ABB RAPID module: 05908a28.mod

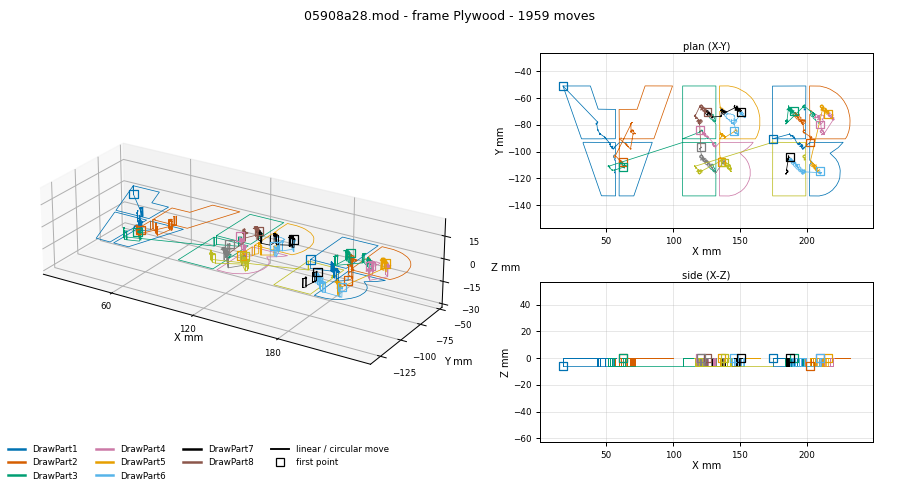
[picture p0: tool path of 05908a28.mod in frame Plywood, 1959 of 1961 moves have a stored position in this frame; points joined in program order, loops and branches not executed]
MODULE ImageDraw
  ! Generated 2026-10-07 09:04 for ABB GoFa CRB 15000-5/0.95: 148 strokes
  ! Page 250 x 180 mm. Work object Plywood: Z points DOWN, so pen-up is -Z and the tool uses orientation [1,0,0,0].
  ! Uses the tool 'tcp' and work object 'Plywood' that already exist on the controller.
  CONST robtarget pOrigin:=[[0,0,0],[1,0,0,0],[0,0,0,0],[9E9,9E9,9E9,9E9,9E9,9E9]];
  CONST jointtarget jHome:=[[0,0,0,0,30,0],[9E9,9E9,9E9,9E9,9E9,9E9]];
  CONST speeddata vTravel:=[250,200,5000,1000];

  PROC DrawImage()
    SingArea\Wrist;
    ConfL\Off;
    ConfJ\Off;
    MoveAbsJ jHome\NoEOffs,vTravel,fine,tcp;
    DrawPart1;
    DrawPart2;
    DrawPart3;
    DrawPart4;
    DrawPart5;
    DrawPart6;
    DrawPart7;
    DrawPart8;
    DrawPart9;
    DrawPart10;
    DrawPart11;
    DrawPart12;
    DrawPart13;
    DrawPart14;
    DrawPart15;
    DrawPart16;
    DrawPart17;
    MoveAbsJ jHome\NoEOffs,vTravel,fine,tcp;
  ENDPROC

  PROC DrawPart1()
    MoveL Offs(pOrigin,17.65,-50.83,-6.00),vTravel,z5,tcp\WObj:=Plywood;
    MoveL Offs(pOrigin,17.65,-50.83,-0.00),v60,z0,tcp\WObj:=Plywood;
    MoveL Offs(pOrigin,38.15,-50.83,-0.00),v40,z0,tcp\WObj:=Plywood;
    MoveL Offs(pOrigin,44.00,-68.18,-0.00),v40,z0,tcp\WObj:=Plywood;
    MoveL Offs(pOrigin,57.00,-68.38,-0.00),v40,z0,tcp\WObj:=Plywood;
    MoveL Offs(pOrigin,56.85,-90.32,-0.00),v40,z0,tcp\WObj:=Plywood;
    MoveL Offs(pOrigin,48.20,-90.38,-0.00),v40,z0,tcp\WObj:=Plywood;
    MoveL Offs(pOrigin,47.75,-90.07,-0.00),v40,z0,tcp\WObj:=Plywood;
    MoveL Offs(pOrigin,47.00,-90.38,-0.00),v40,z0,tcp\WObj:=Plywood;
    MoveL Offs(pOrigin,31.55,-90.38,-0.00),v40,z0,tcp\WObj:=Plywood;
    MoveL Offs(pOrigin,17.65,-50.83,-0.00),v40,fine,tcp\WObj:=Plywood;
    MoveL Offs(pOrigin,17.65,-50.83,-6.00),v60,z5,tcp\WObj:=Plywood;
    MoveL Offs(pOrigin,43.55,-77.82,-6.00),vTravel,z5,tcp\WObj:=Plywood;
    MoveL Offs(pOrigin,43.55,-77.82,-0.00),v60,z0,tcp\WObj:=Plywood;
    MoveL Offs(pOrigin,43.00,-78.68,-0.00),v40,z0,tcp\WObj:=Plywood;
    MoveL Offs(pOrigin,43.85,-77.82,-0.00),v40,z0,tcp\WObj:=Plywood;
    MoveL Offs(pOrigin,43.55,-77.82,-0.00),v40,fine,tcp\WObj:=Plywood;
    MoveL Offs(pOrigin,43.55,-77.82,-6.00),v60,z5,tcp\WObj:=Plywood;
    MoveL Offs(pOrigin,42.95,-78.97,-6.00),vTravel,z5,tcp\WObj:=Plywood;
    MoveL Offs(pOrigin,42.95,-78.97,-0.00),v60,z0,tcp\WObj:=Plywood;
    MoveL Offs(pOrigin,42.65,-78.82,-0.00),v40,z0,tcp\WObj:=Plywood;
    MoveL Offs(pOrigin,42.35,-79.12,-0.00),v40,z0,tcp\WObj:=Plywood;
    MoveL Offs(pOrigin,42.50,-79.43,-0.00),v40,z0,tcp\WObj:=Plywood;
    MoveL Offs(pOrigin,42.95,-78.97,-0.00),v40,z0,tcp\WObj:=Plywood;
    MoveL Offs(pOrigin,42.65,-78.82,-0.00),v40,z0,tcp\WObj:=Plywood;
    MoveL Offs(pOrigin,42.35,-79.28,-0.00),v40,z0,tcp\WObj:=Plywood;
    MoveL Offs(pOrigin,42.95,-78.97,-0.00),v40,fine,tcp\WObj:=Plywood;
    MoveL Offs(pOrigin,42.95,-78.97,-6.00),v60,z5,tcp\WObj:=Plywood;
    MoveL Offs(pOrigin,43.55,-83.78,-6.00),vTravel,z5,tcp\WObj:=Plywood;
    MoveL Offs(pOrigin,43.55,-83.78,-0.00),v60,z0,tcp\WObj:=Plywood;
    MoveL Offs(pOrigin,44.15,-83.78,-0.00),v40,z0,tcp\WObj:=Plywood;
    MoveL Offs(pOrigin,43.55,-83.78,-0.00),v40,fine,tcp\WObj:=Plywood;
    MoveL Offs(pOrigin,43.55,-83.78,-6.00),v60,z5,tcp\WObj:=Plywood;
    MoveL Offs(pOrigin,45.35,-86.62,-6.00),vTravel,z5,tcp\WObj:=Plywood;
    MoveL Offs(pOrigin,45.35,-86.62,-0.00),v60,z0,tcp\WObj:=Plywood;
    MoveL Offs(pOrigin,45.20,-87.07,-0.00),v40,z0,tcp\WObj:=Plywood;
    MoveL Offs(pOrigin,45.65,-86.78,-0.00),v40,z0,tcp\WObj:=Plywood;
    MoveL Offs(pOrigin,45.35,-86.62,-0.00),v40,z0,tcp\WObj:=Plywood;
    MoveL Offs(pOrigin,45.05,-86.93,-0.00),v40,z0,tcp\WObj:=Plywood;
    MoveL Offs(pOrigin,45.35,-87.07,-0.00),v40,z0,tcp\WObj:=Plywood;
    MoveL Offs(pOrigin,45.65,-86.78,-0.00),v40,z0,tcp\WObj:=Plywood;
    MoveL Offs(pOrigin,45.35,-86.62,-0.00),v40,fine,tcp\WObj:=Plywood;
    MoveL Offs(pOrigin,45.35,-86.62,-6.00),v60,z5,tcp\WObj:=Plywood;
    MoveL Offs(pOrigin,48.80,-89.03,-6.00),vTravel,z5,tcp\WObj:=Plywood;
    MoveL Offs(pOrigin,48.80,-89.03,-0.00),v60,z0,tcp\WObj:=Plywood;
    MoveL Offs(pOrigin,48.80,-89.47,-0.00),v40,z0,tcp\WObj:=Plywood;
    MoveL Offs(pOrigin,49.10,-89.32,-0.00),v40,z0,tcp\WObj:=Plywood;
    MoveL Offs(pOrigin,48.95,-89.03,-0.00),v40,z0,tcp\WObj:=Plywood;
    MoveL Offs(pOrigin,48.65,-89.32,-0.00),v40,z0,tcp\WObj:=Plywood;
    MoveL Offs(pOrigin,48.95,-89.47,-0.00),v40,z0,tcp\WObj:=Plywood;
    MoveL Offs(pOrigin,49.10,-89.18,-0.00),v40,z0,tcp\WObj:=Plywood;
    MoveL Offs(pOrigin,48.80,-89.03,-0.00),v40,fine,tcp\WObj:=Plywood;
    MoveL Offs(pOrigin,48.80,-89.03,-6.00),v60,z5,tcp\WObj:=Plywood;
    MoveL Offs(pOrigin,53.00,-94.12,-6.00),vTravel,z5,tcp\WObj:=Plywood;
    MoveL Offs(pOrigin,53.00,-94.12,-0.00),v60,z0,tcp\WObj:=Plywood;
    MoveL Offs(pOrigin,52.55,-94.57,-0.00),v40,z0,tcp\WObj:=Plywood;
    MoveL Offs(pOrigin,52.85,-94.72,-0.00),v40,z0,tcp\WObj:=Plywood;
    MoveL Offs(pOrigin,53.15,-94.28,-0.00),v40,z0,tcp\WObj:=Plywood;
    MoveL Offs(pOrigin,52.55,-94.57,-0.00),v40,z0,tcp\WObj:=Plywood;
    MoveL Offs(pOrigin,52.85,-94.72,-0.00),v40,z0,tcp\WObj:=Plywood;
    MoveL Offs(pOrigin,53.15,-94.43,-0.00),v40,z0,tcp\WObj:=Plywood;
    MoveL Offs(pOrigin,53.00,-94.12,-0.00),v40,fine,tcp\WObj:=Plywood;
    MoveL Offs(pOrigin,53.00,-94.12,-6.00),v60,z5,tcp\WObj:=Plywood;
    MoveL Offs(pOrigin,53.00,-95.93,-6.00),vTravel,z5,tcp\WObj:=Plywood;
    MoveL Offs(pOrigin,53.00,-95.93,-0.00),v60,z0,tcp\WObj:=Plywood;
    MoveL Offs(pOrigin,53.60,-95.93,-0.00),v40,z0,tcp\WObj:=Plywood;
    MoveL Offs(pOrigin,53.00,-95.93,-0.00),v40,fine,tcp\WObj:=Plywood;
    MoveL Offs(pOrigin,53.00,-95.93,-6.00),v60,z5,tcp\WObj:=Plywood;
    MoveL Offs(pOrigin,54.40,-96.53,-6.00),vTravel,z5,tcp\WObj:=Plywood;
    MoveL Offs(pOrigin,54.40,-96.53,-0.00),v60,z0,tcp\WObj:=Plywood;
    MoveL Offs(pOrigin,55.10,-95.82,-0.00),v40,z0,tcp\WObj:=Plywood;
    MoveL Offs(pOrigin,54.65,-95.93,-0.00),v40,z0,tcp\WObj:=Plywood;
    MoveL Offs(pOrigin,54.40,-96.53,-0.00),v40,z0,tcp\WObj:=Plywood;
    MoveL Offs(pOrigin,54.35,-97.43,-0.00),v40,z0,tcp\WObj:=Plywood;
    MoveL Offs(pOrigin,54.35,-96.97,-0.00),v40,z0,tcp\WObj:=Plywood;
    MoveL Offs(pOrigin,54.35,-97.43,-0.00),v40,z0,tcp\WObj:=Plywood;
    MoveL Offs(pOrigin,54.90,-97.72,-0.00),v40,z0,tcp\WObj:=Plywood;
    MoveL Offs(pOrigin,55.25,-98.12,-0.00),v40,z0,tcp\WObj:=Plywood;
    MoveL Offs(pOrigin,55.65,-97.88,-0.00),v40,z0,tcp\WObj:=Plywood;
    MoveL Offs(pOrigin,55.40,-97.57,-0.00),v40,z0,tcp\WObj:=Plywood;
    MoveL Offs(pOrigin,54.90,-97.72,-0.00),v40,fine,tcp\WObj:=Plywood;
    MoveL Offs(pOrigin,54.90,-97.72,-6.00),v60,z5,tcp\WObj:=Plywood;
    MoveL Offs(pOrigin,56.00,-97.12,-6.00),vTravel,z5,tcp\WObj:=Plywood;
    MoveL Offs(pOrigin,56.00,-97.12,-0.00),v60,z0,tcp\WObj:=Plywood;
    MoveL Offs(pOrigin,56.30,-97.38,-0.00),v40,z0,tcp\WObj:=Plywood;
    MoveL Offs(pOrigin,56.90,-96.97,-0.00),v40,z0,tcp\WObj:=Plywood;
    MoveL Offs(pOrigin,56.90,-102.07,-0.00),v40,z0,tcp\WObj:=Plywood;
    MoveL Offs(pOrigin,55.75,-102.68,-0.00),v40,z0,tcp\WObj:=Plywood;
    MoveL Offs(pOrigin,55.40,-103.88,-0.00),v40,z0,tcp\WObj:=Plywood;
    MoveL Offs(pOrigin,55.85,-104.62,-0.00),v40,z0,tcp\WObj:=Plywood;
    MoveL Offs(pOrigin,56.90,-105.07,-0.00),v40,z0,tcp\WObj:=Plywood;
    MoveL Offs(pOrigin,56.15,-106.12,-0.00),v40,z0,tcp\WObj:=Plywood;
    MoveL Offs(pOrigin,56.30,-106.38,-0.00),v40,z0,tcp\WObj:=Plywood;
    MoveL Offs(pOrigin,56.90,-106.28,-0.00),v40,z0,tcp\WObj:=Plywood;
    MoveL Offs(pOrigin,56.90,-113.78,-0.00),v40,z0,tcp\WObj:=Plywood;
    MoveL Offs(pOrigin,56.40,-113.93,-0.00),v40,z0,tcp\WObj:=Plywood;
    MoveL Offs(pOrigin,56.90,-114.68,-0.00),v40,z0,tcp\WObj:=Plywood;
    MoveL Offs(pOrigin,56.70,-115.22,-0.00),v40,z0,tcp\WObj:=Plywood;
    MoveL Offs(pOrigin,56.20,-114.97,-0.00),v40,z0,tcp\WObj:=Plywood;
    MoveL Offs(pOrigin,56.10,-115.88,-0.00),v40,z0,tcp\WObj:=Plywood;
    MoveL Offs(pOrigin,56.85,-115.62,-0.00),v40,z0,tcp\WObj:=Plywood;
    MoveL Offs(pOrigin,57.05,-116.03,-0.00),v40,z0,tcp\WObj:=Plywood;
    MoveL Offs(pOrigin,57.00,-133.07,-0.00),v40,z0,tcp\WObj:=Plywood;
    MoveL Offs(pOrigin,46.45,-132.98,-0.00),v40,z0,tcp\WObj:=Plywood;
    MoveL Offs(pOrigin,32.70,-93.53,-0.00),v40,z0,tcp\WObj:=Plywood;
    MoveL Offs(pOrigin,32.75,-92.97,-0.00),v40,z0,tcp\WObj:=Plywood;
    MoveL Offs(pOrigin,56.90,-93.12,-0.00),v40,z0,tcp\WObj:=Plywood;
    MoveL Offs(pOrigin,56.90,-95.93,-0.00),v40,z0,tcp\WObj:=Plywood;
    MoveL Offs(pOrigin,56.70,-96.32,-0.00),v40,z0,tcp\WObj:=Plywood;
    MoveL Offs(pOrigin,56.20,-96.38,-0.00),v40,z0,tcp\WObj:=Plywood;
    MoveL Offs(pOrigin,56.00,-97.12,-0.00),v40,fine,tcp\WObj:=Plywood;
    MoveL Offs(pOrigin,56.00,-97.12,-6.00),v60,z5,tcp\WObj:=Plywood;
    MoveL Offs(pOrigin,59.80,-93.12,-6.00),vTravel,z5,tcp\WObj:=Plywood;
    MoveL Offs(pOrigin,59.80,-93.12,-0.00),v60,z0,tcp\WObj:=Plywood;
    MoveL Offs(pOrigin,84.45,-92.97,-0.00),v40,z0,tcp\WObj:=Plywood;
    MoveL Offs(pOrigin,70.65,-133.07,-0.00),v40,z0,tcp\WObj:=Plywood;
    MoveL Offs(pOrigin,59.65,-133.07,-0.00),v40,z0,tcp\WObj:=Plywood;
    MoveL Offs(pOrigin,59.75,-108.97,-0.00),v40,z0,tcp\WObj:=Plywood;
    MoveL Offs(pOrigin,60.20,-109.28,-0.00),v40,z0,tcp\WObj:=Plywood;
    MoveL Offs(pOrigin,60.95,-109.18,-0.00),v40,z0,tcp\WObj:=Plywood;
  ENDPROC

  PROC DrawPart2()
    MoveL Offs(pOrigin,62.25,-107.93,-0.00),v40,z0,tcp\WObj:=Plywood;
    MoveL Offs(pOrigin,61.25,-106.72,-0.00),v40,z0,tcp\WObj:=Plywood;
    MoveL Offs(pOrigin,60.65,-106.57,-0.00),v40,z0,tcp\WObj:=Plywood;
    MoveL Offs(pOrigin,60.25,-106.88,-0.00),v40,z0,tcp\WObj:=Plywood;
    MoveL Offs(pOrigin,60.20,-107.62,-0.00),v40,z0,tcp\WObj:=Plywood;
    MoveL Offs(pOrigin,60.75,-108.68,-0.00),v40,z0,tcp\WObj:=Plywood;
    MoveL Offs(pOrigin,59.75,-108.22,-0.00),v40,z0,tcp\WObj:=Plywood;
    MoveL Offs(pOrigin,59.75,-105.93,-0.00),v40,z0,tcp\WObj:=Plywood;
    MoveL Offs(pOrigin,59.90,-106.28,-0.00),v40,z0,tcp\WObj:=Plywood;
    MoveL Offs(pOrigin,60.25,-106.12,-0.00),v40,z0,tcp\WObj:=Plywood;
    MoveL Offs(pOrigin,59.75,-105.22,-0.00),v40,z0,tcp\WObj:=Plywood;
    MoveL Offs(pOrigin,59.80,-93.12,-0.00),v40,fine,tcp\WObj:=Plywood;
    MoveL Offs(pOrigin,59.80,-93.12,-6.00),v60,z5,tcp\WObj:=Plywood;
    MoveL Offs(pOrigin,59.80,-90.32,-6.00),vTravel,z5,tcp\WObj:=Plywood;
    MoveL Offs(pOrigin,59.80,-90.32,-0.00),v60,z0,tcp\WObj:=Plywood;
    MoveL Offs(pOrigin,59.65,-68.38,-0.00),v40,z0,tcp\WObj:=Plywood;
    MoveL Offs(pOrigin,73.10,-68.28,-0.00),v40,z0,tcp\WObj:=Plywood;
    MoveL Offs(pOrigin,79.10,-50.78,-0.00),v40,z0,tcp\WObj:=Plywood;
    MoveL Offs(pOrigin,99.60,-50.83,-0.00),v40,z0,tcp\WObj:=Plywood;
    MoveL Offs(pOrigin,85.65,-90.32,-0.00),v40,z0,tcp\WObj:=Plywood;
    MoveL Offs(pOrigin,61.25,-90.38,-0.00),v40,z0,tcp\WObj:=Plywood;
    MoveL Offs(pOrigin,61.25,-89.68,-0.00),v40,z0,tcp\WObj:=Plywood;
    MoveL Offs(pOrigin,59.80,-90.32,-0.00),v40,fine,tcp\WObj:=Plywood;
    MoveL Offs(pOrigin,59.80,-90.32,-6.00),v60,z5,tcp\WObj:=Plywood;
    MoveL Offs(pOrigin,64.40,-94.12,-6.00),vTravel,z5,tcp\WObj:=Plywood;
    MoveL Offs(pOrigin,64.40,-94.12,-0.00),v60,z0,tcp\WObj:=Plywood;
    MoveL Offs(pOrigin,65.00,-94.12,-0.00),v40,z0,tcp\WObj:=Plywood;
    MoveL Offs(pOrigin,64.40,-94.12,-0.00),v40,z0,tcp\WObj:=Plywood;
    MoveL Offs(pOrigin,65.00,-95.03,-0.00),v40,z0,tcp\WObj:=Plywood;
    MoveL Offs(pOrigin,65.30,-95.32,-0.00),v40,z0,tcp\WObj:=Plywood;
    MoveL Offs(pOrigin,65.60,-95.18,-0.00),v40,z0,tcp\WObj:=Plywood;
    MoveL Offs(pOrigin,65.45,-94.57,-0.00),v40,z0,tcp\WObj:=Plywood;
    MoveL Offs(pOrigin,65.00,-95.03,-0.00),v40,z0,tcp\WObj:=Plywood;
    MoveL Offs(pOrigin,65.30,-95.32,-0.00),v40,z0,tcp\WObj:=Plywood;
    MoveL Offs(pOrigin,65.60,-95.18,-0.00),v40,z0,tcp\WObj:=Plywood;
    MoveL Offs(pOrigin,65.45,-94.57,-0.00),v40,z0,tcp\WObj:=Plywood;
    MoveL Offs(pOrigin,65.00,-95.03,-0.00),v40,fine,tcp\WObj:=Plywood;
    MoveL Offs(pOrigin,65.00,-95.03,-6.00),v60,z5,tcp\WObj:=Plywood;
    MoveL Offs(pOrigin,65.90,-95.93,-6.00),vTravel,z5,tcp\WObj:=Plywood;
    MoveL Offs(pOrigin,65.90,-95.93,-0.00),v60,z0,tcp\WObj:=Plywood;
    MoveL Offs(pOrigin,66.50,-95.93,-0.00),v40,z0,tcp\WObj:=Plywood;
    MoveL Offs(pOrigin,65.90,-95.93,-0.00),v40,fine,tcp\WObj:=Plywood;
    MoveL Offs(pOrigin,65.90,-95.93,-6.00),v60,z5,tcp\WObj:=Plywood;
    MoveL Offs(pOrigin,68.15,-97.88,-6.00),vTravel,z5,tcp\WObj:=Plywood;
    MoveL Offs(pOrigin,68.15,-97.88,-0.00),v60,z0,tcp\WObj:=Plywood;
    MoveL Offs(pOrigin,68.45,-98.03,-0.00),v40,z0,tcp\WObj:=Plywood;
    MoveL Offs(pOrigin,68.60,-97.72,-0.00),v40,z0,tcp\WObj:=Plywood;
    MoveL Offs(pOrigin,68.15,-97.88,-0.00),v40,z0,tcp\WObj:=Plywood;
    MoveL Offs(pOrigin,68.45,-98.03,-0.00),v40,z0,tcp\WObj:=Plywood;
    MoveL Offs(pOrigin,68.45,-97.57,-0.00),v40,z0,tcp\WObj:=Plywood;
    MoveL Offs(pOrigin,68.15,-97.88,-0.00),v40,fine,tcp\WObj:=Plywood;
    MoveL Offs(pOrigin,68.15,-97.88,-6.00),v60,z5,tcp\WObj:=Plywood;
    MoveL Offs(pOrigin,70.10,-86.78,-6.00),vTravel,z5,tcp\WObj:=Plywood;
    MoveL Offs(pOrigin,70.10,-86.78,-0.00),v60,z0,tcp\WObj:=Plywood;
    MoveL Offs(pOrigin,70.55,-86.32,-0.00),v40,z0,tcp\WObj:=Plywood;
    MoveL Offs(pOrigin,70.25,-86.18,-0.00),v40,z0,tcp\WObj:=Plywood;
    MoveL Offs(pOrigin,69.95,-86.62,-0.00),v40,z0,tcp\WObj:=Plywood;
    MoveL Offs(pOrigin,70.55,-86.32,-0.00),v40,z0,tcp\WObj:=Plywood;
    MoveL Offs(pOrigin,70.25,-86.18,-0.00),v40,z0,tcp\WObj:=Plywood;
    MoveL Offs(pOrigin,69.95,-86.47,-0.00),v40,z0,tcp\WObj:=Plywood;
    MoveL Offs(pOrigin,70.10,-86.78,-0.00),v40,fine,tcp\WObj:=Plywood;
    MoveL Offs(pOrigin,70.10,-86.78,-6.00),v60,z5,tcp\WObj:=Plywood;
    MoveL Offs(pOrigin,71.45,-86.47,-6.00),vTravel,z5,tcp\WObj:=Plywood;
    MoveL Offs(pOrigin,71.45,-86.47,-0.00),v60,z0,tcp\WObj:=Plywood;
    MoveL Offs(pOrigin,71.75,-86.62,-0.00),v40,z0,tcp\WObj:=Plywood;
    MoveL Offs(pOrigin,71.90,-86.32,-0.00),v40,z0,tcp\WObj:=Plywood;
    MoveL Offs(pOrigin,71.45,-86.47,-0.00),v40,z0,tcp\WObj:=Plywood;
    MoveL Offs(pOrigin,71.75,-86.62,-0.00),v40,z0,tcp\WObj:=Plywood;
    MoveL Offs(pOrigin,71.75,-86.18,-0.00),v40,z0,tcp\WObj:=Plywood;
    MoveL Offs(pOrigin,71.45,-86.47,-0.00),v40,fine,tcp\WObj:=Plywood;
    MoveL Offs(pOrigin,71.45,-86.47,-6.00),v60,z5,tcp\WObj:=Plywood;
    MoveL Offs(pOrigin,70.50,-84.97,-6.00),vTravel,z5,tcp\WObj:=Plywood;
    MoveL Offs(pOrigin,70.50,-84.97,-0.00),v60,z0,tcp\WObj:=Plywood;
    MoveL Offs(pOrigin,70.50,-84.22,-0.00),v40,z0,tcp\WObj:=Plywood;
    MoveL Offs(pOrigin,69.95,-83.68,-0.00),v40,z0,tcp\WObj:=Plywood;
    MoveL Offs(pOrigin,69.35,-83.62,-0.00),v40,z0,tcp\WObj:=Plywood;
    MoveL Offs(pOrigin,68.75,-84.07,-0.00),v40,z0,tcp\WObj:=Plywood;
    MoveL Offs(pOrigin,68.90,-84.32,-0.00),v40,z0,tcp\WObj:=Plywood;
    MoveL Offs(pOrigin,69.80,-84.03,-0.00),v40,z0,tcp\WObj:=Plywood;
    MoveL Offs(pOrigin,70.50,-84.97,-0.00),v40,fine,tcp\WObj:=Plywood;
    MoveL Offs(pOrigin,70.50,-84.97,-6.00),v60,z5,tcp\WObj:=Plywood;
    MoveL Offs(pOrigin,68.60,-85.47,-6.00),vTravel,z5,tcp\WObj:=Plywood;
    MoveL Offs(pOrigin,68.60,-85.47,-0.00),v60,z0,tcp\WObj:=Plywood;
    MoveL Offs(pOrigin,68.45,-84.47,-0.00),v40,z0,tcp\WObj:=Plywood;
    MoveL Offs(pOrigin,68.15,-84.97,-0.00),v40,z0,tcp\WObj:=Plywood;
    MoveL Offs(pOrigin,68.60,-85.47,-0.00),v40,fine,tcp\WObj:=Plywood;
    MoveL Offs(pOrigin,68.60,-85.47,-6.00),v60,z5,tcp\WObj:=Plywood;
    MoveL Offs(pOrigin,68.45,-79.28,-6.00),vTravel,z5,tcp\WObj:=Plywood;
    MoveL Offs(pOrigin,68.45,-79.28,-0.00),v60,z0,tcp\WObj:=Plywood;
    MoveL Offs(pOrigin,68.75,-78.97,-0.00),v40,z0,tcp\WObj:=Plywood;
    MoveL Offs(pOrigin,68.45,-78.82,-0.00),v40,z0,tcp\WObj:=Plywood;
    MoveL Offs(pOrigin,68.30,-79.28,-0.00),v40,z0,tcp\WObj:=Plywood;
    MoveL Offs(pOrigin,68.75,-78.97,-0.00),v40,z0,tcp\WObj:=Plywood;
    MoveL Offs(pOrigin,68.45,-78.82,-0.00),v40,z0,tcp\WObj:=Plywood;
    MoveL Offs(pOrigin,68.15,-79.12,-0.00),v40,z0,tcp\WObj:=Plywood;
    MoveL Offs(pOrigin,68.45,-79.28,-0.00),v40,fine,tcp\WObj:=Plywood;
    MoveL Offs(pOrigin,68.45,-79.28,-6.00),v60,z5,tcp\WObj:=Plywood;
    MoveL Offs(pOrigin,69.20,-78.07,-6.00),vTravel,z5,tcp\WObj:=Plywood;
    MoveL Offs(pOrigin,69.20,-78.07,-0.00),v60,z0,tcp\WObj:=Plywood;
    MoveL Offs(pOrigin,69.65,-78.07,-0.00),v40,z0,tcp\WObj:=Plywood;
    MoveL Offs(pOrigin,69.20,-78.07,-0.00),v40,fine,tcp\WObj:=Plywood;
    MoveL Offs(pOrigin,69.20,-78.07,-6.00),v60,z5,tcp\WObj:=Plywood;
    MoveL Offs(pOrigin,56.90,-102.97,-6.00),vTravel,z5,tcp\WObj:=Plywood;
    MoveL Offs(pOrigin,56.90,-102.97,-0.00),v60,z0,tcp\WObj:=Plywood;
    MoveL Offs(pOrigin,56.85,-104.43,-0.00),v40,z0,tcp\WObj:=Plywood;
    MoveL Offs(pOrigin,55.85,-103.88,-0.00),v40,z0,tcp\WObj:=Plywood;
    MoveL Offs(pOrigin,55.90,-103.18,-0.00),v40,z0,tcp\WObj:=Plywood;
    MoveL Offs(pOrigin,56.60,-102.82,-0.00),v40,z0,tcp\WObj:=Plywood;
    MoveL Offs(pOrigin,56.90,-102.97,-0.00),v40,fine,tcp\WObj:=Plywood;
    MoveL Offs(pOrigin,56.90,-102.97,-6.00),v60,z5,tcp\WObj:=Plywood;
    MoveL Offs(pOrigin,60.80,-107.22,-6.00),vTravel,z5,tcp\WObj:=Plywood;
    MoveL Offs(pOrigin,60.80,-107.22,-0.00),v60,z0,tcp\WObj:=Plywood;
    MoveL Offs(pOrigin,61.35,-107.47,-0.00),v40,z0,tcp\WObj:=Plywood;
    MoveL Offs(pOrigin,61.25,-108.12,-0.00),v40,z0,tcp\WObj:=Plywood;
    MoveL Offs(pOrigin,60.70,-107.78,-0.00),v40,z0,tcp\WObj:=Plywood;
    MoveL Offs(pOrigin,60.80,-107.22,-0.00),v40,fine,tcp\WObj:=Plywood;
    MoveL Offs(pOrigin,60.80,-107.22,-6.00),v60,z5,tcp\WObj:=Plywood;
    MoveL Offs(pOrigin,62.75,-108.57,-6.00),vTravel,z5,tcp\WObj:=Plywood;
    MoveL Offs(pOrigin,62.75,-108.57,-0.00),v60,z0,tcp\WObj:=Plywood;
    MoveL Offs(pOrigin,61.20,-110.03,-0.00),v40,z0,tcp\WObj:=Plywood;
  ENDPROC

  PROC DrawPart3()
    MoveL Offs(pOrigin,62.45,-111.22,-0.00),v40,z0,tcp\WObj:=Plywood;
    MoveL Offs(pOrigin,63.60,-110.32,-0.00),v40,z0,tcp\WObj:=Plywood;
    MoveL Offs(pOrigin,63.35,-110.12,-0.00),v40,z0,tcp\WObj:=Plywood;
    MoveL Offs(pOrigin,62.45,-110.78,-0.00),v40,z0,tcp\WObj:=Plywood;
    MoveL Offs(pOrigin,62.05,-110.47,-0.00),v40,z0,tcp\WObj:=Plywood;
    MoveL Offs(pOrigin,62.05,-109.72,-0.00),v40,z0,tcp\WObj:=Plywood;
    MoveL Offs(pOrigin,62.85,-108.82,-0.00),v40,z0,tcp\WObj:=Plywood;
    MoveL Offs(pOrigin,62.75,-108.57,-0.00),v40,fine,tcp\WObj:=Plywood;
    MoveL Offs(pOrigin,62.75,-108.57,-6.00),v60,z5,tcp\WObj:=Plywood;
    MoveL Offs(pOrigin,63.80,-109.72,-6.00),vTravel,z5,tcp\WObj:=Plywood;
    MoveL Offs(pOrigin,63.80,-109.72,-0.00),v60,z0,tcp\WObj:=Plywood;
    MoveL Offs(pOrigin,63.50,-110.03,-0.00),v40,z0,tcp\WObj:=Plywood;
    MoveL Offs(pOrigin,63.80,-110.18,-0.00),v40,z0,tcp\WObj:=Plywood;
    MoveL Offs(pOrigin,63.95,-109.88,-0.00),v40,z0,tcp\WObj:=Plywood;
    MoveL Offs(pOrigin,63.50,-110.03,-0.00),v40,z0,tcp\WObj:=Plywood;
    MoveL Offs(pOrigin,63.80,-110.18,-0.00),v40,z0,tcp\WObj:=Plywood;
    MoveL Offs(pOrigin,63.80,-109.72,-0.00),v40,z0,tcp\WObj:=Plywood;
    MoveL Offs(pOrigin,64.40,-110.47,-0.00),v40,z0,tcp\WObj:=Plywood;
    MoveL Offs(pOrigin,63.85,-111.22,-0.00),v40,z0,tcp\WObj:=Plywood;
    MoveL Offs(pOrigin,64.85,-110.88,-0.00),v40,z0,tcp\WObj:=Plywood;
    MoveL Offs(pOrigin,65.10,-110.18,-0.00),v40,z0,tcp\WObj:=Plywood;
    MoveL Offs(pOrigin,64.40,-110.47,-0.00),v40,z0,tcp\WObj:=Plywood;
    MoveL Offs(pOrigin,63.80,-111.32,-0.00),v40,z0,tcp\WObj:=Plywood;
    MoveL Offs(pOrigin,63.15,-111.97,-0.00),v40,z0,tcp\WObj:=Plywood;
    MoveL Offs(pOrigin,63.65,-112.32,-0.00),v40,z0,tcp\WObj:=Plywood;
    MoveL Offs(pOrigin,63.80,-111.32,-0.00),v40,fine,tcp\WObj:=Plywood;
    MoveL Offs(pOrigin,63.80,-111.32,-6.00),v60,z5,tcp\WObj:=Plywood;
    MoveL Offs(pOrigin,56.00,-113.78,-6.00),vTravel,z5,tcp\WObj:=Plywood;
    MoveL Offs(pOrigin,56.00,-113.78,-0.00),v60,z0,tcp\WObj:=Plywood;
    MoveL Offs(pOrigin,56.45,-113.78,-0.00),v40,z0,tcp\WObj:=Plywood;
    MoveL Offs(pOrigin,56.00,-113.78,-0.00),v40,fine,tcp\WObj:=Plywood;
    MoveL Offs(pOrigin,56.00,-113.78,-6.00),v60,z5,tcp\WObj:=Plywood;
    MoveL Offs(pOrigin,54.35,-113.78,-6.00),vTravel,z5,tcp\WObj:=Plywood;
    MoveL Offs(pOrigin,54.35,-113.78,-0.00),v60,z0,tcp\WObj:=Plywood;
    MoveL Offs(pOrigin,54.80,-113.78,-0.00),v40,z0,tcp\WObj:=Plywood;
    MoveL Offs(pOrigin,54.35,-113.78,-0.00),v40,fine,tcp\WObj:=Plywood;
    MoveL Offs(pOrigin,54.35,-113.78,-6.00),v60,z5,tcp\WObj:=Plywood;
    MoveL Offs(pOrigin,52.70,-112.18,-6.00),vTravel,z5,tcp\WObj:=Plywood;
    MoveL Offs(pOrigin,52.70,-112.18,-0.00),v60,z0,tcp\WObj:=Plywood;
    MoveL Offs(pOrigin,52.70,-111.32,-0.00),v40,z0,tcp\WObj:=Plywood;
    MoveL Offs(pOrigin,52.70,-112.18,-0.00),v40,fine,tcp\WObj:=Plywood;
    MoveL Offs(pOrigin,52.70,-112.18,-6.00),v60,z5,tcp\WObj:=Plywood;
    MoveL Offs(pOrigin,51.65,-110.93,-6.00),vTravel,z5,tcp\WObj:=Plywood;
    MoveL Offs(pOrigin,51.65,-110.93,-0.00),v60,z0,tcp\WObj:=Plywood;
    MoveL Offs(pOrigin,51.95,-110.47,-0.00),v40,z0,tcp\WObj:=Plywood;
    MoveL Offs(pOrigin,51.35,-110.78,-0.00),v40,z0,tcp\WObj:=Plywood;
    MoveL Offs(pOrigin,51.65,-110.93,-0.00),v40,z0,tcp\WObj:=Plywood;
    MoveL Offs(pOrigin,51.95,-110.62,-0.00),v40,z0,tcp\WObj:=Plywood;
    MoveL Offs(pOrigin,51.80,-110.32,-0.00),v40,z0,tcp\WObj:=Plywood;
    MoveL Offs(pOrigin,51.35,-110.78,-0.00),v40,z0,tcp\WObj:=Plywood;
    MoveL Offs(pOrigin,51.65,-110.93,-0.00),v40,fine,tcp\WObj:=Plywood;
    MoveL Offs(pOrigin,51.65,-110.93,-6.00),v60,z5,tcp\WObj:=Plywood;
    MoveL Offs(pOrigin,107.20,-93.07,-6.00),vTravel,z5,tcp\WObj:=Plywood;
    MoveL Offs(pOrigin,107.20,-93.07,-0.00),v60,z0,tcp\WObj:=Plywood;
    MoveL Offs(pOrigin,132.00,-93.12,-0.00),v40,z0,tcp\WObj:=Plywood;
    MoveL Offs(pOrigin,132.05,-113.32,-0.00),v40,z0,tcp\WObj:=Plywood;
    MoveL Offs(pOrigin,130.70,-114.32,-0.00),v40,z0,tcp\WObj:=Plywood;
    MoveL Offs(pOrigin,130.30,-114.22,-0.00),v40,z0,tcp\WObj:=Plywood;
    MoveL Offs(pOrigin,130.30,-113.62,-0.00),v40,z0,tcp\WObj:=Plywood;
    MoveL Offs(pOrigin,131.30,-112.43,-0.00),v40,z0,tcp\WObj:=Plywood;
    MoveL Offs(pOrigin,130.60,-112.07,-0.00),v40,z0,tcp\WObj:=Plywood;
    MoveL Offs(pOrigin,130.00,-110.62,-0.00),v40,z0,tcp\WObj:=Plywood;
    MoveL Offs(pOrigin,130.20,-109.72,-0.00),v40,z0,tcp\WObj:=Plywood;
    MoveL Offs(pOrigin,129.65,-109.28,-0.00),v40,z0,tcp\WObj:=Plywood;
    MoveL Offs(pOrigin,127.30,-111.97,-0.00),v40,z0,tcp\WObj:=Plywood;
    MoveL Offs(pOrigin,128.45,-113.22,-0.00),v40,z0,tcp\WObj:=Plywood;
    MoveL Offs(pOrigin,129.45,-113.28,-0.00),v40,z0,tcp\WObj:=Plywood;
    MoveL Offs(pOrigin,129.40,-113.93,-0.00),v40,z0,tcp\WObj:=Plywood;
    MoveL Offs(pOrigin,130.40,-115.03,-0.00),v40,z0,tcp\WObj:=Plywood;
    MoveL Offs(pOrigin,130.85,-115.07,-0.00),v40,z0,tcp\WObj:=Plywood;
    MoveL Offs(pOrigin,131.90,-114.18,-0.00),v40,z0,tcp\WObj:=Plywood;
    MoveL Offs(pOrigin,132.05,-114.38,-0.00),v40,z0,tcp\WObj:=Plywood;
    MoveL Offs(pOrigin,131.45,-114.97,-0.00),v40,z0,tcp\WObj:=Plywood;
    MoveL Offs(pOrigin,131.45,-116.03,-0.00),v40,z0,tcp\WObj:=Plywood;
    MoveL Offs(pOrigin,132.05,-116.78,-0.00),v40,z0,tcp\WObj:=Plywood;
    MoveL Offs(pOrigin,132.00,-133.07,-0.00),v40,z0,tcp\WObj:=Plywood;
    MoveL Offs(pOrigin,107.15,-133.07,-0.00),v40,z0,tcp\WObj:=Plywood;
    MoveL Offs(pOrigin,107.20,-93.07,-0.00),v40,fine,tcp\WObj:=Plywood;
    MoveL Offs(pOrigin,107.20,-93.07,-6.00),v60,z5,tcp\WObj:=Plywood;
    MoveL Offs(pOrigin,107.20,-90.32,-6.00),vTravel,z5,tcp\WObj:=Plywood;
    MoveL Offs(pOrigin,107.20,-90.32,-0.00),v60,z0,tcp\WObj:=Plywood;
    MoveL Offs(pOrigin,107.20,-50.83,-0.00),v40,z0,tcp\WObj:=Plywood;
    MoveL Offs(pOrigin,132.05,-50.83,-0.00),v40,z0,tcp\WObj:=Plywood;
    MoveL Offs(pOrigin,132.05,-75.82,-0.00),v40,z0,tcp\WObj:=Plywood;
    MoveL Offs(pOrigin,130.70,-76.82,-0.00),v40,z0,tcp\WObj:=Plywood;
    MoveL Offs(pOrigin,130.35,-76.72,-0.00),v40,z0,tcp\WObj:=Plywood;
    MoveL Offs(pOrigin,130.30,-76.12,-0.00),v40,z0,tcp\WObj:=Plywood;
    MoveL Offs(pOrigin,131.30,-74.93,-0.00),v40,z0,tcp\WObj:=Plywood;
    MoveL Offs(pOrigin,130.55,-74.47,-0.00),v40,z0,tcp\WObj:=Plywood;
    MoveL Offs(pOrigin,129.90,-72.97,-0.00),v40,z0,tcp\WObj:=Plywood;
    MoveL Offs(pOrigin,130.35,-72.68,-0.00),v40,z0,tcp\WObj:=Plywood;
    MoveL Offs(pOrigin,129.80,-71.93,-0.00),v40,z0,tcp\WObj:=Plywood;
    MoveL Offs(pOrigin,128.45,-72.97,-0.00),v40,z0,tcp\WObj:=Plywood;
    MoveL Offs(pOrigin,127.25,-74.47,-0.00),v40,z0,tcp\WObj:=Plywood;
    MoveL Offs(pOrigin,128.45,-75.72,-0.00),v40,z0,tcp\WObj:=Plywood;
    MoveL Offs(pOrigin,129.45,-75.78,-0.00),v40,z0,tcp\WObj:=Plywood;
    MoveL Offs(pOrigin,129.40,-76.43,-0.00),v40,z0,tcp\WObj:=Plywood;
    MoveL Offs(pOrigin,130.40,-77.57,-0.00),v40,z0,tcp\WObj:=Plywood;
    MoveL Offs(pOrigin,131.00,-77.57,-0.00),v40,z0,tcp\WObj:=Plywood;
    MoveL Offs(pOrigin,132.05,-76.72,-0.00),v40,z0,tcp\WObj:=Plywood;
    MoveL Offs(pOrigin,131.30,-78.07,-0.00),v40,z0,tcp\WObj:=Plywood;
    MoveL Offs(pOrigin,132.05,-79.43,-0.00),v40,z0,tcp\WObj:=Plywood;
    MoveL Offs(pOrigin,132.00,-90.32,-0.00),v40,z0,tcp\WObj:=Plywood;
    MoveL Offs(pOrigin,125.60,-90.28,-0.00),v40,z0,tcp\WObj:=Plywood;
    MoveL Offs(pOrigin,125.80,-89.78,-0.00),v40,z0,tcp\WObj:=Plywood;
    MoveL Offs(pOrigin,125.45,-89.47,-0.00),v40,z0,tcp\WObj:=Plywood;
    MoveL Offs(pOrigin,124.25,-90.38,-0.00),v40,z0,tcp\WObj:=Plywood;
    MoveL Offs(pOrigin,107.20,-90.32,-0.00),v40,fine,tcp\WObj:=Plywood;
    MoveL Offs(pOrigin,107.20,-90.32,-6.00),v60,z5,tcp\WObj:=Plywood;
    MoveL Offs(pOrigin,120.05,-85.32,-6.00),vTravel,z5,tcp\WObj:=Plywood;
    MoveL Offs(pOrigin,120.05,-85.32,-0.00),v60,z0,tcp\WObj:=Plywood;
    MoveL Offs(pOrigin,120.05,-84.62,-0.00),v40,z0,tcp\WObj:=Plywood;
    MoveL Offs(pOrigin,120.05,-85.32,-0.00),v40,fine,tcp\WObj:=Plywood;
    MoveL Offs(pOrigin,120.05,-85.32,-6.00),v60,z5,tcp\WObj:=Plywood;
    MoveL Offs(pOrigin,120.50,-84.18,-6.00),vTravel,z5,tcp\WObj:=Plywood;
    MoveL Offs(pOrigin,120.50,-84.18,-0.00),v60,z0,tcp\WObj:=Plywood;
    MoveL Offs(pOrigin,121.55,-84.12,-0.00),v40,z0,tcp\WObj:=Plywood;
    MoveL Offs(pOrigin,121.85,-84.97,-0.00),v40,z0,tcp\WObj:=Plywood;
    MoveL Offs(pOrigin,122.25,-84.82,-0.00),v40,z0,tcp\WObj:=Plywood;
    MoveL Offs(pOrigin,121.55,-83.68,-0.00),v40,z0,tcp\WObj:=Plywood;
  ENDPROC

  PROC DrawPart4()
    MoveL Offs(pOrigin,120.40,-83.93,-0.00),v40,z0,tcp\WObj:=Plywood;
    MoveL Offs(pOrigin,120.50,-84.18,-0.00),v40,fine,tcp\WObj:=Plywood;
    MoveL Offs(pOrigin,120.50,-84.18,-6.00),v60,z5,tcp\WObj:=Plywood;
    MoveL Offs(pOrigin,122.30,-85.57,-6.00),vTravel,z5,tcp\WObj:=Plywood;
    MoveL Offs(pOrigin,122.30,-85.57,-0.00),v60,z0,tcp\WObj:=Plywood;
    MoveL Offs(pOrigin,121.85,-86.43,-0.00),v40,z0,tcp\WObj:=Plywood;
    MoveL Offs(pOrigin,122.40,-86.18,-0.00),v40,z0,tcp\WObj:=Plywood;
    MoveL Offs(pOrigin,122.90,-85.32,-0.00),v40,z0,tcp\WObj:=Plywood;
    MoveL Offs(pOrigin,122.30,-85.57,-0.00),v40,z0,tcp\WObj:=Plywood;
    MoveL Offs(pOrigin,122.75,-86.47,-0.00),v40,z0,tcp\WObj:=Plywood;
    MoveL Offs(pOrigin,122.20,-87.38,-0.00),v40,z0,tcp\WObj:=Plywood;
    MoveL Offs(pOrigin,123.00,-87.07,-0.00),v40,z0,tcp\WObj:=Plywood;
    MoveL Offs(pOrigin,123.20,-86.38,-0.00),v40,z0,tcp\WObj:=Plywood;
    MoveL Offs(pOrigin,122.75,-86.47,-0.00),v40,z0,tcp\WObj:=Plywood;
    MoveL Offs(pOrigin,123.20,-87.07,-0.00),v40,z0,tcp\WObj:=Plywood;
    MoveL Offs(pOrigin,123.05,-87.38,-0.00),v40,z0,tcp\WObj:=Plywood;
    MoveL Offs(pOrigin,123.50,-87.82,-0.00),v40,z0,tcp\WObj:=Plywood;
    MoveL Offs(pOrigin,123.65,-87.53,-0.00),v40,z0,tcp\WObj:=Plywood;
    MoveL Offs(pOrigin,123.05,-87.22,-0.00),v40,z0,tcp\WObj:=Plywood;
    MoveL Offs(pOrigin,123.50,-87.82,-0.00),v40,z0,tcp\WObj:=Plywood;
    MoveL Offs(pOrigin,123.65,-87.53,-0.00),v40,z0,tcp\WObj:=Plywood;
    MoveL Offs(pOrigin,123.20,-87.07,-0.00),v40,z0,tcp\WObj:=Plywood;
    MoveL Offs(pOrigin,123.80,-86.68,-0.00),v40,z0,tcp\WObj:=Plywood;
    MoveL Offs(pOrigin,124.20,-86.62,-0.00),v40,z0,tcp\WObj:=Plywood;
    MoveL Offs(pOrigin,123.95,-86.28,-0.00),v40,z0,tcp\WObj:=Plywood;
    MoveL Offs(pOrigin,123.55,-86.32,-0.00),v40,z0,tcp\WObj:=Plywood;
    MoveL Offs(pOrigin,123.80,-86.68,-0.00),v40,z0,tcp\WObj:=Plywood;
    MoveL Offs(pOrigin,124.10,-86.78,-0.00),v40,z0,tcp\WObj:=Plywood;
    MoveL Offs(pOrigin,124.40,-87.38,-0.00),v40,z0,tcp\WObj:=Plywood;
    MoveL Offs(pOrigin,124.55,-86.93,-0.00),v40,z0,tcp\WObj:=Plywood;
    MoveL Offs(pOrigin,124.25,-86.62,-0.00),v40,z0,tcp\WObj:=Plywood;
    MoveL Offs(pOrigin,124.40,-87.38,-0.00),v40,z0,tcp\WObj:=Plywood;
    MoveL Offs(pOrigin,124.55,-86.93,-0.00),v40,z0,tcp\WObj:=Plywood;
    MoveL Offs(pOrigin,124.10,-86.78,-0.00),v40,z0,tcp\WObj:=Plywood;
    MoveL Offs(pOrigin,123.80,-87.82,-0.00),v40,z0,tcp\WObj:=Plywood;
    MoveL Offs(pOrigin,123.55,-87.82,-0.00),v40,z0,tcp\WObj:=Plywood;
    MoveL Offs(pOrigin,123.50,-88.38,-0.00),v40,z0,tcp\WObj:=Plywood;
    MoveL Offs(pOrigin,123.95,-88.28,-0.00),v40,z0,tcp\WObj:=Plywood;
    MoveL Offs(pOrigin,123.80,-87.82,-0.00),v40,fine,tcp\WObj:=Plywood;
    MoveL Offs(pOrigin,123.80,-87.82,-6.00),v60,z5,tcp\WObj:=Plywood;
    MoveL Offs(pOrigin,124.70,-88.72,-6.00),vTravel,z5,tcp\WObj:=Plywood;
    MoveL Offs(pOrigin,124.70,-88.72,-0.00),v60,z0,tcp\WObj:=Plywood;
    MoveL Offs(pOrigin,125.75,-88.38,-0.00),v40,z0,tcp\WObj:=Plywood;
    MoveL Offs(pOrigin,125.75,-88.12,-0.00),v40,z0,tcp\WObj:=Plywood;
    MoveL Offs(pOrigin,125.15,-87.93,-0.00),v40,z0,tcp\WObj:=Plywood;
    MoveL Offs(pOrigin,124.70,-88.72,-0.00),v40,fine,tcp\WObj:=Plywood;
    MoveL Offs(pOrigin,124.70,-88.72,-6.00),v60,z5,tcp\WObj:=Plywood;
    MoveL Offs(pOrigin,126.10,-88.88,-6.00),vTravel,z5,tcp\WObj:=Plywood;
    MoveL Offs(pOrigin,126.10,-88.88,-0.00),v60,z0,tcp\WObj:=Plywood;
    MoveL Offs(pOrigin,125.95,-89.47,-0.00),v40,z0,tcp\WObj:=Plywood;
    MoveL Offs(pOrigin,126.60,-89.03,-0.00),v40,z0,tcp\WObj:=Plywood;
    MoveL Offs(pOrigin,126.10,-88.88,-0.00),v40,fine,tcp\WObj:=Plywood;
    MoveL Offs(pOrigin,126.10,-88.88,-6.00),v60,z5,tcp\WObj:=Plywood;
    MoveL Offs(pOrigin,129.95,-93.28,-6.00),vTravel,z5,tcp\WObj:=Plywood;
    MoveL Offs(pOrigin,129.95,-93.28,-0.00),v60,z0,tcp\WObj:=Plywood;
    MoveL Offs(pOrigin,129.20,-94.22,-0.00),v40,z0,tcp\WObj:=Plywood;
    MoveL Offs(pOrigin,129.65,-94.12,-0.00),v40,z0,tcp\WObj:=Plywood;
    MoveL Offs(pOrigin,130.20,-93.38,-0.00),v40,z0,tcp\WObj:=Plywood;
    MoveL Offs(pOrigin,129.95,-93.28,-0.00),v40,z0,tcp\WObj:=Plywood;
    MoveL Offs(pOrigin,130.55,-93.82,-0.00),v40,z0,tcp\WObj:=Plywood;
    MoveL Offs(pOrigin,130.70,-94.12,-0.00),v40,z0,tcp\WObj:=Plywood;
    MoveL Offs(pOrigin,131.00,-93.68,-0.00),v40,z0,tcp\WObj:=Plywood;
    MoveL Offs(pOrigin,130.55,-93.82,-0.00),v40,z0,tcp\WObj:=Plywood;
    MoveL Offs(pOrigin,130.70,-94.12,-0.00),v40,z0,tcp\WObj:=Plywood;
    MoveL Offs(pOrigin,131.00,-93.82,-0.00),v40,z0,tcp\WObj:=Plywood;
    MoveL Offs(pOrigin,130.85,-93.53,-0.00),v40,z0,tcp\WObj:=Plywood;
    MoveL Offs(pOrigin,130.55,-93.82,-0.00),v40,z0,tcp\WObj:=Plywood;
    MoveL Offs(pOrigin,130.40,-93.97,-0.00),v40,z0,tcp\WObj:=Plywood;
    MoveL Offs(pOrigin,130.40,-94.43,-0.00),v40,z0,tcp\WObj:=Plywood;
    MoveL Offs(pOrigin,130.70,-94.12,-0.00),v40,z0,tcp\WObj:=Plywood;
    MoveL Offs(pOrigin,130.40,-93.97,-0.00),v40,z0,tcp\WObj:=Plywood;
    MoveL Offs(pOrigin,130.25,-94.28,-0.00),v40,z0,tcp\WObj:=Plywood;
    MoveL Offs(pOrigin,130.70,-94.12,-0.00),v40,z0,tcp\WObj:=Plywood;
    MoveL Offs(pOrigin,130.40,-93.97,-0.00),v40,z0,tcp\WObj:=Plywood;
    MoveL Offs(pOrigin,130.10,-94.72,-0.00),v40,z0,tcp\WObj:=Plywood;
    MoveL Offs(pOrigin,129.80,-94.57,-0.00),v40,z0,tcp\WObj:=Plywood;
    MoveL Offs(pOrigin,129.80,-95.18,-0.00),v40,z0,tcp\WObj:=Plywood;
    MoveL Offs(pOrigin,130.10,-94.72,-0.00),v40,z0,tcp\WObj:=Plywood;
    MoveL Offs(pOrigin,129.80,-94.57,-0.00),v40,z0,tcp\WObj:=Plywood;
    MoveL Offs(pOrigin,129.65,-95.03,-0.00),v40,z0,tcp\WObj:=Plywood;
    MoveL Offs(pOrigin,130.10,-94.72,-0.00),v40,fine,tcp\WObj:=Plywood;
    MoveL Offs(pOrigin,130.10,-94.72,-6.00),v60,z5,tcp\WObj:=Plywood;
    MoveL Offs(pOrigin,130.40,-95.93,-6.00),vTravel,z5,tcp\WObj:=Plywood;
    MoveL Offs(pOrigin,130.40,-95.93,-0.00),v60,z0,tcp\WObj:=Plywood;
    MoveL Offs(pOrigin,131.00,-95.93,-0.00),v40,z0,tcp\WObj:=Plywood;
    MoveL Offs(pOrigin,130.40,-95.93,-0.00),v40,fine,tcp\WObj:=Plywood;
    MoveL Offs(pOrigin,130.40,-95.93,-6.00),v60,z5,tcp\WObj:=Plywood;
    MoveL Offs(pOrigin,131.45,-95.32,-6.00),vTravel,z5,tcp\WObj:=Plywood;
    MoveL Offs(pOrigin,131.45,-95.32,-0.00),v60,z0,tcp\WObj:=Plywood;
    MoveL Offs(pOrigin,131.75,-95.47,-0.00),v40,z0,tcp\WObj:=Plywood;
    MoveL Offs(pOrigin,131.90,-95.18,-0.00),v40,z0,tcp\WObj:=Plywood;
    MoveL Offs(pOrigin,131.45,-95.18,-0.00),v40,z0,tcp\WObj:=Plywood;
    MoveL Offs(pOrigin,131.75,-95.47,-0.00),v40,z0,tcp\WObj:=Plywood;
    MoveL Offs(pOrigin,131.75,-95.03,-0.00),v40,z0,tcp\WObj:=Plywood;
    MoveL Offs(pOrigin,131.45,-95.32,-0.00),v40,z0,tcp\WObj:=Plywood;
    MoveL Offs(pOrigin,131.75,-96.47,-0.00),v40,z0,tcp\WObj:=Plywood;
    MoveL Offs(pOrigin,131.45,-96.82,-0.00),v40,z0,tcp\WObj:=Plywood;
    MoveL Offs(pOrigin,131.75,-97.47,-0.00),v40,z0,tcp\WObj:=Plywood;
    MoveL Offs(pOrigin,131.75,-96.47,-0.00),v40,fine,tcp\WObj:=Plywood;
    MoveL Offs(pOrigin,131.75,-96.47,-6.00),v60,z5,tcp\WObj:=Plywood;
    MoveL Offs(pOrigin,134.90,-93.12,-6.00),vTravel,z5,tcp\WObj:=Plywood;
    MoveL Offs(pOrigin,134.90,-93.12,-0.00),v60,z0,tcp\WObj:=Plywood;
    MoveL Offs(pOrigin,159.95,-92.97,-0.00),v40,z0,tcp\WObj:=Plywood;
    MoveL Offs(pOrigin,158.45,-94.88,-0.00),v40,z0,tcp\WObj:=Plywood;
    MoveL Offs(pOrigin,155.30,-97.72,-0.00),v40,z0,tcp\WObj:=Plywood;
    MoveL Offs(pOrigin,150.15,-101.18,-0.00),v40,z0,tcp\WObj:=Plywood;
    MoveL Offs(pOrigin,153.95,-104.78,-0.00),v40,z0,tcp\WObj:=Plywood;
    MoveL Offs(pOrigin,155.15,-106.43,-0.00),v40,z0,tcp\WObj:=Plywood;
    MoveL Offs(pOrigin,156.55,-109.12,-0.00),v40,z0,tcp\WObj:=Plywood;
    MoveL Offs(pOrigin,157.70,-113.32,-0.00),v40,z0,tcp\WObj:=Plywood;
    MoveL Offs(pOrigin,157.70,-117.97,-0.00),v40,z0,tcp\WObj:=Plywood;
    MoveL Offs(pOrigin,156.85,-121.28,-0.00),v40,z0,tcp\WObj:=Plywood;
    MoveL Offs(pOrigin,155.20,-124.72,-0.00),v40,z0,tcp\WObj:=Plywood;
    MoveL Offs(pOrigin,153.35,-127.28,-0.00),v40,z0,tcp\WObj:=Plywood;
    MoveL Offs(pOrigin,150.95,-129.52,-0.00),v40,z0,tcp\WObj:=Plywood;
    MoveL Offs(pOrigin,146.30,-132.12,-0.00),v40,z0,tcp\WObj:=Plywood;
    MoveL Offs(pOrigin,141.95,-133.12,-0.00),v40,z0,tcp\WObj:=Plywood;
    MoveL Offs(pOrigin,134.75,-133.07,-0.00),v40,z0,tcp\WObj:=Plywood;
    MoveL Offs(pOrigin,134.90,-106.53,-0.00),v40,z0,tcp\WObj:=Plywood;
    MoveL Offs(pOrigin,135.20,-107.18,-0.00),v40,z0,tcp\WObj:=Plywood;
  ENDPROC

  PROC DrawPart5()
    MoveL Offs(pOrigin,136.25,-107.47,-0.00),v40,z0,tcp\WObj:=Plywood;
    MoveL Offs(pOrigin,137.10,-106.72,-0.00),v40,z0,tcp\WObj:=Plywood;
    MoveL Offs(pOrigin,136.15,-105.53,-0.00),v40,z0,tcp\WObj:=Plywood;
    MoveL Offs(pOrigin,136.85,-105.62,-0.00),v40,z0,tcp\WObj:=Plywood;
    MoveL Offs(pOrigin,137.15,-106.53,-0.00),v40,z0,tcp\WObj:=Plywood;
    MoveL Offs(pOrigin,137.60,-106.12,-0.00),v40,z0,tcp\WObj:=Plywood;
    MoveL Offs(pOrigin,137.00,-105.07,-0.00),v40,z0,tcp\WObj:=Plywood;
    MoveL Offs(pOrigin,136.25,-104.78,-0.00),v40,z0,tcp\WObj:=Plywood;
    MoveL Offs(pOrigin,135.00,-105.72,-0.00),v40,z0,tcp\WObj:=Plywood;
    MoveL Offs(pOrigin,135.85,-104.32,-0.00),v40,z0,tcp\WObj:=Plywood;
    MoveL Offs(pOrigin,135.50,-104.12,-0.00),v40,z0,tcp\WObj:=Plywood;
    MoveL Offs(pOrigin,134.95,-104.43,-0.00),v40,z0,tcp\WObj:=Plywood;
    MoveL Offs(pOrigin,135.20,-103.12,-0.00),v40,z0,tcp\WObj:=Plywood;
    MoveL Offs(pOrigin,134.90,-102.53,-0.00),v40,z0,tcp\WObj:=Plywood;
    MoveL Offs(pOrigin,134.90,-93.12,-0.00),v40,fine,tcp\WObj:=Plywood;
    MoveL Offs(pOrigin,134.90,-93.12,-6.00),v60,z5,tcp\WObj:=Plywood;
    MoveL Offs(pOrigin,134.95,-90.32,-6.00),vTravel,z5,tcp\WObj:=Plywood;
    MoveL Offs(pOrigin,134.95,-90.32,-0.00),v60,z0,tcp\WObj:=Plywood;
    MoveL Offs(pOrigin,134.90,-86.78,-0.00),v40,z0,tcp\WObj:=Plywood;
    MoveL Offs(pOrigin,135.60,-85.57,-0.00),v40,z0,tcp\WObj:=Plywood;
    MoveL Offs(pOrigin,134.90,-85.72,-0.00),v40,z0,tcp\WObj:=Plywood;
    MoveL Offs(pOrigin,135.20,-84.82,-0.00),v40,z0,tcp\WObj:=Plywood;
    MoveL Offs(pOrigin,134.90,-83.47,-0.00),v40,z0,tcp\WObj:=Plywood;
    MoveL Offs(pOrigin,134.95,-74.78,-0.00),v40,z0,tcp\WObj:=Plywood;
    MoveL Offs(pOrigin,135.30,-74.62,-0.00),v40,z0,tcp\WObj:=Plywood;
    MoveL Offs(pOrigin,134.90,-74.03,-0.00),v40,z0,tcp\WObj:=Plywood;
    MoveL Offs(pOrigin,134.90,-69.82,-0.00),v40,z0,tcp\WObj:=Plywood;
    MoveL Offs(pOrigin,136.70,-69.88,-0.00),v40,z0,tcp\WObj:=Plywood;
    MoveL Offs(pOrigin,137.75,-68.47,-0.00),v40,z0,tcp\WObj:=Plywood;
    MoveL Offs(pOrigin,137.15,-67.57,-0.00),v40,z0,tcp\WObj:=Plywood;
    MoveL Offs(pOrigin,136.40,-67.28,-0.00),v40,z0,tcp\WObj:=Plywood;
    MoveL Offs(pOrigin,135.25,-67.68,-0.00),v40,z0,tcp\WObj:=Plywood;
    MoveL Offs(pOrigin,135.80,-66.97,-0.00),v40,z0,tcp\WObj:=Plywood;
    MoveL Offs(pOrigin,135.65,-66.57,-0.00),v40,z0,tcp\WObj:=Plywood;
    MoveL Offs(pOrigin,134.95,-66.93,-0.00),v40,z0,tcp\WObj:=Plywood;
    MoveL Offs(pOrigin,135.20,-66.22,-0.00),v40,z0,tcp\WObj:=Plywood;
    MoveL Offs(pOrigin,134.75,-61.58,-0.00),v40,z0,tcp\WObj:=Plywood;
    MoveL Offs(pOrigin,134.75,-50.83,-0.00),v40,z0,tcp\WObj:=Plywood;
    MoveL Offs(pOrigin,141.35,-50.78,-0.00),v40,z0,tcp\WObj:=Plywood;
    MoveL Offs(pOrigin,146.00,-51.67,-0.00),v40,z0,tcp\WObj:=Plywood;
    MoveL Offs(pOrigin,148.85,-52.67,-0.00),v40,z0,tcp\WObj:=Plywood;
    MoveL Offs(pOrigin,154.55,-55.88,-0.00),v40,z0,tcp\WObj:=Plywood;
    MoveL Offs(pOrigin,158.45,-59.47,-0.00),v40,z0,tcp\WObj:=Plywood;
    MoveL Offs(pOrigin,160.10,-61.58,-0.00),v40,z0,tcp\WObj:=Plywood;
    MoveL Offs(pOrigin,163.00,-66.82,-0.00),v40,z0,tcp\WObj:=Plywood;
    MoveL Offs(pOrigin,164.00,-69.82,-0.00),v40,z0,tcp\WObj:=Plywood;
    MoveL Offs(pOrigin,164.90,-74.32,-0.00),v40,z0,tcp\WObj:=Plywood;
    MoveL Offs(pOrigin,164.90,-80.62,-0.00),v40,z0,tcp\WObj:=Plywood;
    MoveL Offs(pOrigin,164.45,-83.47,-0.00),v40,z0,tcp\WObj:=Plywood;
    MoveL Offs(pOrigin,163.00,-87.97,-0.00),v40,z0,tcp\WObj:=Plywood;
    MoveL Offs(pOrigin,161.60,-90.38,-0.00),v40,z0,tcp\WObj:=Plywood;
    MoveL Offs(pOrigin,138.65,-90.38,-0.00),v40,z0,tcp\WObj:=Plywood;
    MoveL Offs(pOrigin,138.05,-90.07,-0.00),v40,z0,tcp\WObj:=Plywood;
    MoveL Offs(pOrigin,137.30,-90.38,-0.00),v40,z0,tcp\WObj:=Plywood;
    MoveL Offs(pOrigin,134.95,-90.32,-0.00),v40,fine,tcp\WObj:=Plywood;
    MoveL Offs(pOrigin,134.95,-90.32,-6.00),v60,z5,tcp\WObj:=Plywood;
    MoveL Offs(pOrigin,136.55,-88.43,-6.00),vTravel,z5,tcp\WObj:=Plywood;
    MoveL Offs(pOrigin,136.55,-88.43,-0.00),v60,z0,tcp\WObj:=Plywood;
    MoveL Offs(pOrigin,136.85,-88.12,-0.00),v40,z0,tcp\WObj:=Plywood;
    MoveL Offs(pOrigin,136.70,-87.68,-0.00),v40,z0,tcp\WObj:=Plywood;
    MoveL Offs(pOrigin,136.40,-87.82,-0.00),v40,z0,tcp\WObj:=Plywood;
    MoveL Offs(pOrigin,136.55,-88.43,-0.00),v40,z0,tcp\WObj:=Plywood;
    MoveL Offs(pOrigin,136.85,-87.82,-0.00),v40,z0,tcp\WObj:=Plywood;
    MoveL Offs(pOrigin,136.40,-87.82,-0.00),v40,z0,tcp\WObj:=Plywood;
    MoveL Offs(pOrigin,136.55,-88.43,-0.00),v40,z0,tcp\WObj:=Plywood;
    MoveL Offs(pOrigin,136.40,-87.82,-0.00),v40,z0,tcp\WObj:=Plywood;
    MoveL Offs(pOrigin,136.55,-87.53,-0.00),v40,z0,tcp\WObj:=Plywood;
    MoveL Offs(pOrigin,136.10,-87.22,-0.00),v40,z0,tcp\WObj:=Plywood;
    MoveL Offs(pOrigin,136.40,-87.82,-0.00),v40,z0,tcp\WObj:=Plywood;
    MoveL Offs(pOrigin,136.55,-87.53,-0.00),v40,z0,tcp\WObj:=Plywood;
    MoveL Offs(pOrigin,136.25,-87.22,-0.00),v40,z0,tcp\WObj:=Plywood;
    MoveL Offs(pOrigin,135.95,-87.38,-0.00),v40,z0,tcp\WObj:=Plywood;
    MoveL Offs(pOrigin,136.40,-87.82,-0.00),v40,z0,tcp\WObj:=Plywood;
    MoveL Offs(pOrigin,135.80,-87.18,-0.00),v40,z0,tcp\WObj:=Plywood;
    MoveL Offs(pOrigin,136.35,-86.32,-0.00),v40,z0,tcp\WObj:=Plywood;
    MoveL Offs(pOrigin,135.50,-86.47,-0.00),v40,z0,tcp\WObj:=Plywood;
    MoveL Offs(pOrigin,135.40,-87.07,-0.00),v40,z0,tcp\WObj:=Plywood;
    MoveL Offs(pOrigin,135.80,-87.18,-0.00),v40,z0,tcp\WObj:=Plywood;
    MoveL Offs(pOrigin,136.55,-86.38,-0.00),v40,z0,tcp\WObj:=Plywood;
    MoveL Offs(pOrigin,137.40,-87.53,-0.00),v40,z0,tcp\WObj:=Plywood;
    MoveL Offs(pOrigin,137.10,-86.47,-0.00),v40,z0,tcp\WObj:=Plywood;
    MoveL Offs(pOrigin,136.55,-86.38,-0.00),v40,fine,tcp\WObj:=Plywood;
    MoveL Offs(pOrigin,136.55,-86.38,-6.00),v60,z5,tcp\WObj:=Plywood;
    MoveL Offs(pOrigin,137.90,-87.97,-6.00),vTravel,z5,tcp\WObj:=Plywood;
    MoveL Offs(pOrigin,137.90,-87.97,-0.00),v60,z0,tcp\WObj:=Plywood;
    MoveL Offs(pOrigin,137.90,-88.43,-0.00),v40,z0,tcp\WObj:=Plywood;
    MoveL Offs(pOrigin,138.35,-88.12,-0.00),v40,z0,tcp\WObj:=Plywood;
    MoveL Offs(pOrigin,137.90,-87.97,-0.00),v40,z0,tcp\WObj:=Plywood;
    MoveL Offs(pOrigin,137.75,-88.28,-0.00),v40,z0,tcp\WObj:=Plywood;
    MoveL Offs(pOrigin,138.05,-88.43,-0.00),v40,z0,tcp\WObj:=Plywood;
    MoveL Offs(pOrigin,138.35,-88.12,-0.00),v40,z0,tcp\WObj:=Plywood;
    MoveL Offs(pOrigin,137.90,-87.97,-0.00),v40,fine,tcp\WObj:=Plywood;
    MoveL Offs(pOrigin,137.90,-87.97,-6.00),v60,z5,tcp\WObj:=Plywood;
    MoveL Offs(pOrigin,139.10,-88.88,-6.00),vTravel,z5,tcp\WObj:=Plywood;
    MoveL Offs(pOrigin,139.10,-88.88,-0.00),v60,z0,tcp\WObj:=Plywood;
    MoveL Offs(pOrigin,138.80,-89.32,-0.00),v40,z0,tcp\WObj:=Plywood;
    MoveL Offs(pOrigin,139.10,-89.47,-0.00),v40,z0,tcp\WObj:=Plywood;
    MoveL Offs(pOrigin,139.40,-89.18,-0.00),v40,z0,tcp\WObj:=Plywood;
    MoveL Offs(pOrigin,139.10,-88.88,-0.00),v40,z0,tcp\WObj:=Plywood;
    MoveL Offs(pOrigin,138.80,-89.32,-0.00),v40,z0,tcp\WObj:=Plywood;
    MoveL Offs(pOrigin,139.10,-89.47,-0.00),v40,z0,tcp\WObj:=Plywood;
    MoveL Offs(pOrigin,139.40,-89.18,-0.00),v40,z0,tcp\WObj:=Plywood;
    MoveL Offs(pOrigin,139.10,-88.88,-0.00),v40,z0,tcp\WObj:=Plywood;
    MoveL Offs(pOrigin,138.50,-89.47,-0.00),v40,z0,tcp\WObj:=Plywood;
    MoveL Offs(pOrigin,138.20,-89.78,-0.00),v40,z0,tcp\WObj:=Plywood;
    MoveL Offs(pOrigin,138.35,-90.18,-0.00),v40,z0,tcp\WObj:=Plywood;
    MoveL Offs(pOrigin,138.80,-89.78,-0.00),v40,z0,tcp\WObj:=Plywood;
    MoveL Offs(pOrigin,138.50,-89.47,-0.00),v40,fine,tcp\WObj:=Plywood;
    MoveL Offs(pOrigin,138.50,-89.47,-6.00),v60,z5,tcp\WObj:=Plywood;
    MoveL Offs(pOrigin,145.55,-85.12,-6.00),vTravel,z5,tcp\WObj:=Plywood;
    MoveL Offs(pOrigin,145.55,-85.12,-0.00),v60,z0,tcp\WObj:=Plywood;
    MoveL Offs(pOrigin,146.00,-85.72,-0.00),v40,z0,tcp\WObj:=Plywood;
    MoveL Offs(pOrigin,146.25,-85.72,-0.00),v40,z0,tcp\WObj:=Plywood;
    MoveL Offs(pOrigin,146.10,-84.68,-0.00),v40,z0,tcp\WObj:=Plywood;
    MoveL Offs(pOrigin,146.60,-84.12,-0.00),v40,z0,tcp\WObj:=Plywood;
    MoveL Offs(pOrigin,147.35,-84.12,-0.00),v40,z0,tcp\WObj:=Plywood;
    MoveL Offs(pOrigin,147.90,-84.97,-0.00),v40,z0,tcp\WObj:=Plywood;
    MoveL Offs(pOrigin,147.90,-84.22,-0.00),v40,z0,tcp\WObj:=Plywood;
    MoveL Offs(pOrigin,147.20,-83.53,-0.00),v40,z0,tcp\WObj:=Plywood;
    MoveL Offs(pOrigin,146.30,-83.72,-0.00),v40,z0,tcp\WObj:=Plywood;
  ENDPROC

  PROC DrawPart6()
    MoveL Offs(pOrigin,145.60,-84.53,-0.00),v40,z0,tcp\WObj:=Plywood;
    MoveL Offs(pOrigin,145.55,-85.12,-0.00),v40,z0,tcp\WObj:=Plywood;
    MoveL Offs(pOrigin,146.30,-85.88,-0.00),v40,z0,tcp\WObj:=Plywood;
    MoveL Offs(pOrigin,147.05,-85.88,-0.00),v40,z0,tcp\WObj:=Plywood;
    MoveL Offs(pOrigin,146.30,-85.88,-0.00),v40,fine,tcp\WObj:=Plywood;
    MoveL Offs(pOrigin,146.30,-85.88,-6.00),v60,z5,tcp\WObj:=Plywood;
    MoveL Offs(pOrigin,147.35,-86.47,-6.00),vTravel,z5,tcp\WObj:=Plywood;
    MoveL Offs(pOrigin,147.35,-86.47,-0.00),v60,z0,tcp\WObj:=Plywood;
    MoveL Offs(pOrigin,147.80,-86.32,-0.00),v40,z0,tcp\WObj:=Plywood;
    MoveL Offs(pOrigin,147.50,-86.18,-0.00),v40,z0,tcp\WObj:=Plywood;
    MoveL Offs(pOrigin,147.50,-86.62,-0.00),v40,z0,tcp\WObj:=Plywood;
    MoveL Offs(pOrigin,147.80,-86.32,-0.00),v40,z0,tcp\WObj:=Plywood;
    MoveL Offs(pOrigin,147.50,-86.18,-0.00),v40,z0,tcp\WObj:=Plywood;
    MoveL Offs(pOrigin,147.35,-86.47,-0.00),v40,z0,tcp\WObj:=Plywood;
    MoveL Offs(pOrigin,148.25,-86.78,-0.00),v40,z0,tcp\WObj:=Plywood;
    MoveL Offs(pOrigin,148.40,-87.07,-0.00),v40,z0,tcp\WObj:=Plywood;
    MoveL Offs(pOrigin,148.70,-86.93,-0.00),v40,z0,tcp\WObj:=Plywood;
    MoveL Offs(pOrigin,148.55,-86.47,-0.00),v40,z0,tcp\WObj:=Plywood;
    MoveL Offs(pOrigin,148.25,-86.93,-0.00),v40,z0,tcp\WObj:=Plywood;
    MoveL Offs(pOrigin,148.70,-86.93,-0.00),v40,z0,tcp\WObj:=Plywood;
    MoveL Offs(pOrigin,148.55,-86.47,-0.00),v40,z0,tcp\WObj:=Plywood;
    MoveL Offs(pOrigin,148.25,-86.78,-0.00),v40,fine,tcp\WObj:=Plywood;
    MoveL Offs(pOrigin,148.25,-86.78,-6.00),v60,z5,tcp\WObj:=Plywood;
    MoveL Offs(pOrigin,145.70,-79.68,-6.00),vTravel,z5,tcp\WObj:=Plywood;
    MoveL Offs(pOrigin,145.70,-79.68,-0.00),v60,z0,tcp\WObj:=Plywood;
    MoveL Offs(pOrigin,147.80,-77.32,-0.00),v40,z0,tcp\WObj:=Plywood;
    MoveL Offs(pOrigin,147.05,-75.93,-0.00),v40,z0,tcp\WObj:=Plywood;
    MoveL Offs(pOrigin,146.30,-75.72,-0.00),v40,z0,tcp\WObj:=Plywood;
    MoveL Offs(pOrigin,145.60,-76.28,-0.00),v40,z0,tcp\WObj:=Plywood;
    MoveL Offs(pOrigin,145.45,-75.38,-0.00),v40,z0,tcp\WObj:=Plywood;
    MoveL Offs(pOrigin,146.00,-75.18,-0.00),v40,z0,tcp\WObj:=Plywood;
    MoveL Offs(pOrigin,146.25,-74.62,-0.00),v40,z0,tcp\WObj:=Plywood;
    MoveL Offs(pOrigin,146.15,-73.78,-0.00),v40,z0,tcp\WObj:=Plywood;
    MoveL Offs(pOrigin,145.55,-73.43,-0.00),v40,z0,tcp\WObj:=Plywood;
    MoveL Offs(pOrigin,146.10,-72.97,-0.00),v40,z0,tcp\WObj:=Plywood;
    MoveL Offs(pOrigin,145.25,-72.68,-0.00),v40,z0,tcp\WObj:=Plywood;
    MoveL Offs(pOrigin,144.80,-72.07,-0.00),v40,z0,tcp\WObj:=Plywood;
    MoveL Offs(pOrigin,143.60,-72.07,-0.00),v40,z0,tcp\WObj:=Plywood;
    MoveL Offs(pOrigin,142.85,-71.62,-0.00),v40,z0,tcp\WObj:=Plywood;
    MoveL Offs(pOrigin,141.80,-71.88,-0.00),v40,z0,tcp\WObj:=Plywood;
    MoveL Offs(pOrigin,141.35,-71.47,-0.00),v40,z0,tcp\WObj:=Plywood;
    MoveL Offs(pOrigin,139.60,-72.78,-0.00),v40,z0,tcp\WObj:=Plywood;
    MoveL Offs(pOrigin,140.65,-71.18,-0.00),v40,z0,tcp\WObj:=Plywood;
    MoveL Offs(pOrigin,140.45,-70.72,-0.00),v40,z0,tcp\WObj:=Plywood;
    MoveL Offs(pOrigin,140.00,-70.62,-0.00),v40,z0,tcp\WObj:=Plywood;
    MoveL Offs(pOrigin,138.35,-72.22,-0.00),v40,z0,tcp\WObj:=Plywood;
    MoveL Offs(pOrigin,138.25,-72.68,-0.00),v40,z0,tcp\WObj:=Plywood;
    MoveL Offs(pOrigin,139.25,-73.88,-0.00),v40,z0,tcp\WObj:=Plywood;
    MoveL Offs(pOrigin,140.10,-73.93,-0.00),v40,z0,tcp\WObj:=Plywood;
    MoveL Offs(pOrigin,139.70,-74.78,-0.00),v40,z0,tcp\WObj:=Plywood;
    MoveL Offs(pOrigin,139.85,-75.07,-0.00),v40,z0,tcp\WObj:=Plywood;
    MoveL Offs(pOrigin,140.30,-75.18,-0.00),v40,z0,tcp\WObj:=Plywood;
    MoveL Offs(pOrigin,140.45,-74.82,-0.00),v40,z0,tcp\WObj:=Plywood;
    MoveL Offs(pOrigin,141.35,-76.07,-0.00),v40,z0,tcp\WObj:=Plywood;
    MoveL Offs(pOrigin,142.15,-75.88,-0.00),v40,z0,tcp\WObj:=Plywood;
    MoveL Offs(pOrigin,141.90,-76.43,-0.00),v40,z0,tcp\WObj:=Plywood;
    MoveL Offs(pOrigin,142.90,-77.62,-0.00),v40,z0,tcp\WObj:=Plywood;
    MoveL Offs(pOrigin,144.00,-77.72,-0.00),v40,z0,tcp\WObj:=Plywood;
    MoveL Offs(pOrigin,144.35,-78.97,-0.00),v40,z0,tcp\WObj:=Plywood;
    MoveL Offs(pOrigin,145.70,-79.68,-0.00),v40,z0,tcp\WObj:=Plywood;
    MoveL Offs(pOrigin,145.40,-78.62,-0.00),v40,z0,tcp\WObj:=Plywood;
    MoveL Offs(pOrigin,145.30,-77.93,-0.00),v40,z0,tcp\WObj:=Plywood;
    MoveL Offs(pOrigin,145.85,-77.47,-0.00),v40,z0,tcp\WObj:=Plywood;
    MoveL Offs(pOrigin,145.90,-78.22,-0.00),v40,z0,tcp\WObj:=Plywood;
    MoveL Offs(pOrigin,145.40,-78.62,-0.00),v40,fine,tcp\WObj:=Plywood;
    MoveL Offs(pOrigin,145.40,-78.62,-6.00),v60,z5,tcp\WObj:=Plywood;
    MoveL Offs(pOrigin,144.05,-78.68,-6.00),vTravel,z5,tcp\WObj:=Plywood;
    MoveL Offs(pOrigin,144.05,-78.68,-0.00),v60,z0,tcp\WObj:=Plywood;
    MoveL Offs(pOrigin,143.90,-78.28,-0.00),v40,z0,tcp\WObj:=Plywood;
    MoveL Offs(pOrigin,143.60,-78.53,-0.00),v40,z0,tcp\WObj:=Plywood;
    MoveL Offs(pOrigin,143.75,-78.93,-0.00),v40,z0,tcp\WObj:=Plywood;
    MoveL Offs(pOrigin,144.05,-78.68,-0.00),v40,fine,tcp\WObj:=Plywood;
    MoveL Offs(pOrigin,144.05,-78.68,-6.00),v60,z5,tcp\WObj:=Plywood;
    MoveL Offs(pOrigin,143.45,-76.57,-6.00),vTravel,z5,tcp\WObj:=Plywood;
    MoveL Offs(pOrigin,143.45,-76.57,-0.00),v60,z0,tcp\WObj:=Plywood;
    MoveL Offs(pOrigin,143.35,-76.18,-0.00),v40,z0,tcp\WObj:=Plywood;
    MoveL Offs(pOrigin,143.95,-76.18,-0.00),v40,z0,tcp\WObj:=Plywood;
    MoveL Offs(pOrigin,143.45,-76.57,-0.00),v40,fine,tcp\WObj:=Plywood;
    MoveL Offs(pOrigin,143.45,-76.57,-6.00),v60,z5,tcp\WObj:=Plywood;
    MoveL Offs(pOrigin,146.75,-77.03,-6.00),vTravel,z5,tcp\WObj:=Plywood;
    MoveL Offs(pOrigin,146.75,-77.03,-0.00),v60,z0,tcp\WObj:=Plywood;
    MoveL Offs(pOrigin,146.30,-76.72,-0.00),v40,z0,tcp\WObj:=Plywood;
    MoveL Offs(pOrigin,146.75,-77.03,-0.00),v40,fine,tcp\WObj:=Plywood;
    MoveL Offs(pOrigin,146.75,-77.03,-6.00),v60,z5,tcp\WObj:=Plywood;
    MoveL Offs(pOrigin,150.65,-71.93,-6.00),vTravel,z5,tcp\WObj:=Plywood;
    MoveL Offs(pOrigin,150.65,-71.93,-0.00),v60,z0,tcp\WObj:=Plywood;
    MoveL Offs(pOrigin,152.20,-70.43,-0.00),v40,z0,tcp\WObj:=Plywood;
    MoveL Offs(pOrigin,151.85,-70.28,-0.00),v40,z0,tcp\WObj:=Plywood;
    MoveL Offs(pOrigin,150.65,-71.18,-0.00),v40,z0,tcp\WObj:=Plywood;
    MoveL Offs(pOrigin,150.05,-70.22,-0.00),v40,z0,tcp\WObj:=Plywood;
    MoveL Offs(pOrigin,149.65,-70.88,-0.00),v40,z0,tcp\WObj:=Plywood;
    MoveL Offs(pOrigin,150.65,-71.93,-0.00),v40,z0,tcp\WObj:=Plywood;
    MoveL Offs(pOrigin,151.45,-72.38,-0.00),v40,z0,tcp\WObj:=Plywood;
    MoveL Offs(pOrigin,151.85,-73.07,-0.00),v40,z0,tcp\WObj:=Plywood;
    MoveL Offs(pOrigin,152.90,-71.22,-0.00),v40,z0,tcp\WObj:=Plywood;
    MoveL Offs(pOrigin,151.45,-72.38,-0.00),v40,z0,tcp\WObj:=Plywood;
    MoveL Offs(pOrigin,152.10,-73.28,-0.00),v40,z0,tcp\WObj:=Plywood;
    MoveL Offs(pOrigin,152.75,-73.72,-0.00),v40,z0,tcp\WObj:=Plywood;
    MoveL Offs(pOrigin,153.40,-73.12,-0.00),v40,z0,tcp\WObj:=Plywood;
    MoveL Offs(pOrigin,152.10,-73.28,-0.00),v40,fine,tcp\WObj:=Plywood;
    MoveL Offs(pOrigin,152.10,-73.28,-6.00),v60,z5,tcp\WObj:=Plywood;
    MoveL Offs(pOrigin,153.35,-74.32,-6.00),vTravel,z5,tcp\WObj:=Plywood;
    MoveL Offs(pOrigin,153.35,-74.32,-0.00),v60,z0,tcp\WObj:=Plywood;
    MoveL Offs(pOrigin,153.80,-74.62,-0.00),v40,z0,tcp\WObj:=Plywood;
    MoveL Offs(pOrigin,153.80,-74.03,-0.00),v40,z0,tcp\WObj:=Plywood;
    MoveL Offs(pOrigin,153.35,-74.47,-0.00),v40,z0,tcp\WObj:=Plywood;
    MoveL Offs(pOrigin,153.80,-74.62,-0.00),v40,z0,tcp\WObj:=Plywood;
    MoveL Offs(pOrigin,153.95,-74.18,-0.00),v40,z0,tcp\WObj:=Plywood;
    MoveL Offs(pOrigin,153.65,-74.03,-0.00),v40,z0,tcp\WObj:=Plywood;
    MoveL Offs(pOrigin,153.35,-74.32,-0.00),v40,fine,tcp\WObj:=Plywood;
    MoveL Offs(pOrigin,153.35,-74.32,-6.00),v60,z5,tcp\WObj:=Plywood;
    MoveL Offs(pOrigin,150.95,-70.72,-6.00),vTravel,z5,tcp\WObj:=Plywood;
    MoveL Offs(pOrigin,150.95,-70.72,-0.00),v60,z0,tcp\WObj:=Plywood;
    MoveL Offs(pOrigin,151.10,-70.43,-0.00),v40,z0,tcp\WObj:=Plywood;
    MoveL Offs(pOrigin,150.80,-70.12,-0.00),v40,z0,tcp\WObj:=Plywood;
    MoveL Offs(pOrigin,150.65,-70.43,-0.00),v40,z0,tcp\WObj:=Plywood;
    MoveL Offs(pOrigin,151.10,-70.57,-0.00),v40,z0,tcp\WObj:=Plywood;
    MoveL Offs(pOrigin,150.80,-70.12,-0.00),v40,z0,tcp\WObj:=Plywood;
    MoveL Offs(pOrigin,150.65,-70.43,-0.00),v40,z0,tcp\WObj:=Plywood;
    MoveL Offs(pOrigin,150.95,-70.72,-0.00),v40,z0,tcp\WObj:=Plywood;
  ENDPROC

  PROC DrawPart7()
    MoveL Offs(pOrigin,150.50,-70.12,-0.00),v40,z0,tcp\WObj:=Plywood;
    MoveL Offs(pOrigin,151.25,-69.22,-0.00),v40,z0,tcp\WObj:=Plywood;
    MoveL Offs(pOrigin,150.50,-69.53,-0.00),v40,z0,tcp\WObj:=Plywood;
    MoveL Offs(pOrigin,150.50,-70.12,-0.00),v40,z0,tcp\WObj:=Plywood;
    MoveL Offs(pOrigin,149.90,-69.38,-0.00),v40,z0,tcp\WObj:=Plywood;
    MoveL Offs(pOrigin,148.85,-67.57,-0.00),v40,z0,tcp\WObj:=Plywood;
    MoveL Offs(pOrigin,148.25,-67.88,-0.00),v40,z0,tcp\WObj:=Plywood;
    MoveL Offs(pOrigin,147.80,-68.62,-0.00),v40,z0,tcp\WObj:=Plywood;
    MoveL Offs(pOrigin,147.90,-69.22,-0.00),v40,z0,tcp\WObj:=Plywood;
    MoveL Offs(pOrigin,148.70,-69.97,-0.00),v40,z0,tcp\WObj:=Plywood;
    MoveL Offs(pOrigin,149.60,-69.78,-0.00),v40,z0,tcp\WObj:=Plywood;
    MoveL Offs(pOrigin,149.90,-69.38,-0.00),v40,z0,tcp\WObj:=Plywood;
    MoveL Offs(pOrigin,150.20,-68.68,-0.00),v40,z0,tcp\WObj:=Plywood;
    MoveL Offs(pOrigin,150.35,-68.32,-0.00),v40,z0,tcp\WObj:=Plywood;
    MoveL Offs(pOrigin,150.05,-67.97,-0.00),v40,z0,tcp\WObj:=Plywood;
    MoveL Offs(pOrigin,149.90,-68.32,-0.00),v40,z0,tcp\WObj:=Plywood;
    MoveL Offs(pOrigin,150.20,-68.68,-0.00),v40,fine,tcp\WObj:=Plywood;
    MoveL Offs(pOrigin,150.20,-68.68,-6.00),v60,z5,tcp\WObj:=Plywood;
    MoveL Offs(pOrigin,149.00,-68.78,-6.00),vTravel,z5,tcp\WObj:=Plywood;
    MoveL Offs(pOrigin,149.00,-68.78,-0.00),v60,z0,tcp\WObj:=Plywood;
    MoveL Offs(pOrigin,149.10,-69.32,-0.00),v40,z0,tcp\WObj:=Plywood;
    MoveL Offs(pOrigin,148.50,-69.07,-0.00),v40,z0,tcp\WObj:=Plywood;
    MoveL Offs(pOrigin,148.55,-68.53,-0.00),v40,z0,tcp\WObj:=Plywood;
    MoveL Offs(pOrigin,149.00,-68.78,-0.00),v40,fine,tcp\WObj:=Plywood;
    MoveL Offs(pOrigin,149.00,-68.78,-6.00),v60,z5,tcp\WObj:=Plywood;
    MoveL Offs(pOrigin,146.90,-68.93,-6.00),vTravel,z5,tcp\WObj:=Plywood;
    MoveL Offs(pOrigin,146.90,-68.93,-0.00),v60,z0,tcp\WObj:=Plywood;
    MoveL Offs(pOrigin,148.65,-66.68,-0.00),v40,z0,tcp\WObj:=Plywood;
    MoveL Offs(pOrigin,148.40,-66.57,-0.00),v40,z0,tcp\WObj:=Plywood;
    MoveL Offs(pOrigin,147.05,-67.72,-0.00),v40,z0,tcp\WObj:=Plywood;
    MoveL Offs(pOrigin,146.20,-68.93,-0.00),v40,z0,tcp\WObj:=Plywood;
    MoveL Offs(pOrigin,146.90,-68.93,-0.00),v40,fine,tcp\WObj:=Plywood;
    MoveL Offs(pOrigin,146.90,-68.93,-6.00),v60,z5,tcp\WObj:=Plywood;
    MoveL Offs(pOrigin,146.75,-67.43,-6.00),vTravel,z5,tcp\WObj:=Plywood;
    MoveL Offs(pOrigin,146.75,-67.43,-0.00),v60,z0,tcp\WObj:=Plywood;
    MoveL Offs(pOrigin,147.00,-66.97,-0.00),v40,z0,tcp\WObj:=Plywood;
    MoveL Offs(pOrigin,146.00,-66.38,-0.00),v40,z0,tcp\WObj:=Plywood;
    MoveL Offs(pOrigin,146.35,-65.32,-0.00),v40,z0,tcp\WObj:=Plywood;
    MoveL Offs(pOrigin,146.15,-65.22,-0.00),v40,z0,tcp\WObj:=Plywood;
    MoveL Offs(pOrigin,145.55,-66.38,-0.00),v40,z0,tcp\WObj:=Plywood;
    MoveL Offs(pOrigin,146.00,-67.12,-0.00),v40,z0,tcp\WObj:=Plywood;
    MoveL Offs(pOrigin,146.75,-67.43,-0.00),v40,fine,tcp\WObj:=Plywood;
    MoveL Offs(pOrigin,146.75,-67.43,-6.00),v60,z5,tcp\WObj:=Plywood;
    MoveL Offs(pOrigin,147.80,-66.38,-6.00),vTravel,z5,tcp\WObj:=Plywood;
    MoveL Offs(pOrigin,147.80,-66.38,-0.00),v60,z0,tcp\WObj:=Plywood;
    MoveL Offs(pOrigin,147.80,-65.78,-0.00),v40,z0,tcp\WObj:=Plywood;
    MoveL Offs(pOrigin,147.80,-66.38,-0.00),v40,fine,tcp\WObj:=Plywood;
    MoveL Offs(pOrigin,147.80,-66.38,-6.00),v60,z5,tcp\WObj:=Plywood;
    MoveL Offs(pOrigin,140.00,-70.28,-6.00),vTravel,z5,tcp\WObj:=Plywood;
    MoveL Offs(pOrigin,140.00,-70.28,-0.00),v60,z0,tcp\WObj:=Plywood;
    MoveL Offs(pOrigin,138.20,-68.88,-0.00),v40,z0,tcp\WObj:=Plywood;
    MoveL Offs(pOrigin,137.60,-69.22,-0.00),v40,z0,tcp\WObj:=Plywood;
    MoveL Offs(pOrigin,137.35,-69.82,-0.00),v40,z0,tcp\WObj:=Plywood;
    MoveL Offs(pOrigin,137.85,-71.12,-0.00),v40,z0,tcp\WObj:=Plywood;
    MoveL Offs(pOrigin,137.30,-70.03,-0.00),v40,z0,tcp\WObj:=Plywood;
    MoveL Offs(pOrigin,136.85,-70.03,-0.00),v40,z0,tcp\WObj:=Plywood;
    MoveL Offs(pOrigin,136.60,-70.57,-0.00),v40,z0,tcp\WObj:=Plywood;
    MoveL Offs(pOrigin,137.20,-71.93,-0.00),v40,z0,tcp\WObj:=Plywood;
    MoveL Offs(pOrigin,138.05,-72.07,-0.00),v40,z0,tcp\WObj:=Plywood;
    MoveL Offs(pOrigin,140.00,-70.28,-0.00),v40,fine,tcp\WObj:=Plywood;
    MoveL Offs(pOrigin,140.00,-70.28,-6.00),v60,z5,tcp\WObj:=Plywood;
    MoveL Offs(pOrigin,138.65,-70.43,-6.00),vTravel,z5,tcp\WObj:=Plywood;
    MoveL Offs(pOrigin,138.65,-70.43,-0.00),v60,z0,tcp\WObj:=Plywood;
    MoveL Offs(pOrigin,138.35,-70.43,-0.00),v40,z0,tcp\WObj:=Plywood;
    MoveL Offs(pOrigin,138.20,-69.97,-0.00),v40,z0,tcp\WObj:=Plywood;
    MoveL Offs(pOrigin,138.50,-69.97,-0.00),v40,z0,tcp\WObj:=Plywood;
    MoveL Offs(pOrigin,138.65,-70.43,-0.00),v40,z0,tcp\WObj:=Plywood;
    MoveL Offs(pOrigin,138.20,-70.12,-0.00),v40,z0,tcp\WObj:=Plywood;
    MoveL Offs(pOrigin,138.50,-69.97,-0.00),v40,z0,tcp\WObj:=Plywood;
    MoveL Offs(pOrigin,138.65,-70.43,-0.00),v40,fine,tcp\WObj:=Plywood;
    MoveL Offs(pOrigin,138.65,-70.43,-6.00),v60,z5,tcp\WObj:=Plywood;
    MoveL Offs(pOrigin,136.80,-68.82,-6.00),vTravel,z5,tcp\WObj:=Plywood;
    MoveL Offs(pOrigin,136.80,-68.82,-0.00),v60,z0,tcp\WObj:=Plywood;
    MoveL Offs(pOrigin,136.25,-67.97,-0.00),v40,z0,tcp\WObj:=Plywood;
    MoveL Offs(pOrigin,136.80,-68.18,-0.00),v40,z0,tcp\WObj:=Plywood;
    MoveL Offs(pOrigin,136.80,-68.82,-0.00),v40,z0,tcp\WObj:=Plywood;
    MoveL Offs(pOrigin,136.10,-69.22,-0.00),v40,z0,tcp\WObj:=Plywood;
    MoveL Offs(pOrigin,135.65,-69.22,-0.00),v40,z0,tcp\WObj:=Plywood;
    MoveL Offs(pOrigin,135.50,-68.93,-0.00),v40,z0,tcp\WObj:=Plywood;
    MoveL Offs(pOrigin,135.80,-68.78,-0.00),v40,z0,tcp\WObj:=Plywood;
    MoveL Offs(pOrigin,136.10,-69.22,-0.00),v40,z0,tcp\WObj:=Plywood;
    MoveL Offs(pOrigin,135.50,-68.93,-0.00),v40,z0,tcp\WObj:=Plywood;
    MoveL Offs(pOrigin,135.80,-68.78,-0.00),v40,z0,tcp\WObj:=Plywood;
    MoveL Offs(pOrigin,136.10,-69.22,-0.00),v40,fine,tcp\WObj:=Plywood;
    MoveL Offs(pOrigin,136.10,-69.22,-6.00),v60,z5,tcp\WObj:=Plywood;
    MoveL Offs(pOrigin,135.95,-73.57,-6.00),vTravel,z5,tcp\WObj:=Plywood;
    MoveL Offs(pOrigin,135.95,-73.57,-0.00),v60,z0,tcp\WObj:=Plywood;
    MoveL Offs(pOrigin,135.95,-72.82,-0.00),v40,z0,tcp\WObj:=Plywood;
    MoveL Offs(pOrigin,135.95,-73.57,-0.00),v40,fine,tcp\WObj:=Plywood;
    MoveL Offs(pOrigin,135.95,-73.57,-6.00),v60,z5,tcp\WObj:=Plywood;
    MoveL Offs(pOrigin,129.50,-74.03,-6.00),vTravel,z5,tcp\WObj:=Plywood;
    MoveL Offs(pOrigin,129.50,-74.03,-0.00),v60,z0,tcp\WObj:=Plywood;
    MoveL Offs(pOrigin,129.35,-74.88,-0.00),v40,z0,tcp\WObj:=Plywood;
    MoveL Offs(pOrigin,128.60,-74.78,-0.00),v40,z0,tcp\WObj:=Plywood;
    MoveL Offs(pOrigin,128.60,-74.18,-0.00),v40,z0,tcp\WObj:=Plywood;
    MoveL Offs(pOrigin,129.50,-74.03,-0.00),v40,fine,tcp\WObj:=Plywood;
    MoveL Offs(pOrigin,129.50,-74.03,-6.00),v60,z5,tcp\WObj:=Plywood;
    MoveL Offs(pOrigin,128.85,-72.07,-6.00),vTravel,z5,tcp\WObj:=Plywood;
    MoveL Offs(pOrigin,128.85,-72.07,-0.00),v60,z0,tcp\WObj:=Plywood;
    MoveL Offs(pOrigin,128.15,-71.82,-0.00),v40,z0,tcp\WObj:=Plywood;
    MoveL Offs(pOrigin,126.85,-72.93,-0.00),v40,z0,tcp\WObj:=Plywood;
    MoveL Offs(pOrigin,126.70,-72.38,-0.00),v40,z0,tcp\WObj:=Plywood;
    MoveL Offs(pOrigin,127.65,-71.03,-0.00),v40,z0,tcp\WObj:=Plywood;
    MoveL Offs(pOrigin,126.05,-69.22,-0.00),v40,z0,tcp\WObj:=Plywood;
    MoveL Offs(pOrigin,125.00,-68.97,-0.00),v40,z0,tcp\WObj:=Plywood;
    MoveL Offs(pOrigin,123.85,-70.28,-0.00),v40,z0,tcp\WObj:=Plywood;
    MoveL Offs(pOrigin,123.85,-71.18,-0.00),v40,z0,tcp\WObj:=Plywood;
    MoveL Offs(pOrigin,125.15,-72.18,-0.00),v40,z0,tcp\WObj:=Plywood;
    MoveL Offs(pOrigin,126.75,-70.93,-0.00),v40,z0,tcp\WObj:=Plywood;
    MoveL Offs(pOrigin,125.35,-72.53,-0.00),v40,z0,tcp\WObj:=Plywood;
    MoveL Offs(pOrigin,126.50,-73.82,-0.00),v40,z0,tcp\WObj:=Plywood;
    MoveL Offs(pOrigin,127.40,-73.82,-0.00),v40,z0,tcp\WObj:=Plywood;
    MoveL Offs(pOrigin,128.85,-72.07,-0.00),v40,fine,tcp\WObj:=Plywood;
    MoveL Offs(pOrigin,128.85,-72.07,-6.00),v60,z5,tcp\WObj:=Plywood;
    MoveL Offs(pOrigin,125.60,-70.57,-6.00),vTravel,z5,tcp\WObj:=Plywood;
    MoveL Offs(pOrigin,125.60,-70.57,-0.00),v60,z0,tcp\WObj:=Plywood;
    MoveL Offs(pOrigin,125.30,-69.82,-0.00),v40,z0,tcp\WObj:=Plywood;
    MoveL Offs(pOrigin,125.75,-70.12,-0.00),v40,z0,tcp\WObj:=Plywood;
    MoveL Offs(pOrigin,125.60,-70.57,-0.00),v40,z0,tcp\WObj:=Plywood;
    MoveL Offs(pOrigin,125.30,-69.82,-0.00),v40,z0,tcp\WObj:=Plywood;
  ENDPROC

  PROC DrawPart8()
    MoveL Offs(pOrigin,125.75,-70.12,-0.00),v40,z0,tcp\WObj:=Plywood;
    MoveL Offs(pOrigin,125.60,-70.57,-0.00),v40,z0,tcp\WObj:=Plywood;
    MoveL Offs(pOrigin,124.85,-70.57,-0.00),v40,z0,tcp\WObj:=Plywood;
    MoveL Offs(pOrigin,124.55,-70.72,-0.00),v40,z0,tcp\WObj:=Plywood;
    MoveL Offs(pOrigin,124.55,-70.28,-0.00),v40,z0,tcp\WObj:=Plywood;
    MoveL Offs(pOrigin,124.85,-70.72,-0.00),v40,z0,tcp\WObj:=Plywood;
    MoveL Offs(pOrigin,124.55,-70.72,-0.00),v40,z0,tcp\WObj:=Plywood;
    MoveL Offs(pOrigin,124.55,-70.28,-0.00),v40,z0,tcp\WObj:=Plywood;
    MoveL Offs(pOrigin,124.85,-70.57,-0.00),v40,fine,tcp\WObj:=Plywood;
    MoveL Offs(pOrigin,124.85,-70.57,-6.00),v60,z5,tcp\WObj:=Plywood;
    MoveL Offs(pOrigin,123.65,-70.03,-6.00),vTravel,z5,tcp\WObj:=Plywood;
    MoveL Offs(pOrigin,123.65,-70.03,-0.00),v60,z0,tcp\WObj:=Plywood;
    MoveL Offs(pOrigin,124.80,-68.93,-0.00),v40,z0,tcp\WObj:=Plywood;
    MoveL Offs(pOrigin,124.80,-68.18,-0.00),v40,z0,tcp\WObj:=Plywood;
    MoveL Offs(pOrigin,123.95,-67.32,-0.00),v40,z0,tcp\WObj:=Plywood;
    MoveL Offs(pOrigin,122.75,-67.47,-0.00),v40,z0,tcp\WObj:=Plywood;
    MoveL Offs(pOrigin,122.05,-68.32,-0.00),v40,z0,tcp\WObj:=Plywood;
    MoveL Offs(pOrigin,122.10,-69.38,-0.00),v40,z0,tcp\WObj:=Plywood;
    MoveL Offs(pOrigin,122.60,-69.93,-0.00),v40,z0,tcp\WObj:=Plywood;
    MoveL Offs(pOrigin,123.65,-70.03,-0.00),v40,z0,tcp\WObj:=Plywood;
    MoveL Offs(pOrigin,123.20,-69.22,-0.00),v40,z0,tcp\WObj:=Plywood;
    MoveL Offs(pOrigin,122.80,-69.18,-0.00),v40,z0,tcp\WObj:=Plywood;
    MoveL Offs(pOrigin,122.80,-68.72,-0.00),v40,z0,tcp\WObj:=Plywood;
    MoveL Offs(pOrigin,123.20,-69.22,-0.00),v40,z0,tcp\WObj:=Plywood;
    MoveL Offs(pOrigin,124.05,-68.88,-0.00),v40,z0,tcp\WObj:=Plywood;
    MoveL Offs(pOrigin,123.25,-68.18,-0.00),v40,z0,tcp\WObj:=Plywood;
    MoveL Offs(pOrigin,123.35,-67.93,-0.00),v40,z0,tcp\WObj:=Plywood;
    MoveL Offs(pOrigin,123.95,-68.32,-0.00),v40,z0,tcp\WObj:=Plywood;
    MoveL Offs(pOrigin,124.05,-68.88,-0.00),v40,fine,tcp\WObj:=Plywood;
    MoveL Offs(pOrigin,124.05,-68.88,-6.00),v60,z5,tcp\WObj:=Plywood;
    MoveL Offs(pOrigin,123.00,-66.82,-6.00),vTravel,z5,tcp\WObj:=Plywood;
    MoveL Offs(pOrigin,123.00,-66.82,-0.00),v60,z0,tcp\WObj:=Plywood;
    MoveL Offs(pOrigin,122.90,-66.53,-0.00),v40,z0,tcp\WObj:=Plywood;
    MoveL Offs(pOrigin,122.15,-66.82,-0.00),v40,z0,tcp\WObj:=Plywood;
    MoveL Offs(pOrigin,120.55,-68.78,-0.00),v40,z0,tcp\WObj:=Plywood;
    MoveL Offs(pOrigin,120.95,-68.88,-0.00),v40,z0,tcp\WObj:=Plywood;
    MoveL Offs(pOrigin,123.00,-66.82,-0.00),v40,z0,tcp\WObj:=Plywood;
    MoveL Offs(pOrigin,122.00,-66.47,-0.00),v40,z0,tcp\WObj:=Plywood;
    MoveL Offs(pOrigin,122.30,-65.93,-0.00),v40,z0,tcp\WObj:=Plywood;
    MoveL Offs(pOrigin,121.70,-65.22,-0.00),v40,z0,tcp\WObj:=Plywood;
    MoveL Offs(pOrigin,121.70,-66.22,-0.00),v40,z0,tcp\WObj:=Plywood;
    MoveL Offs(pOrigin,122.00,-66.47,-0.00),v40,z0,tcp\WObj:=Plywood;
    MoveL Offs(pOrigin,121.25,-66.88,-0.00),v40,z0,tcp\WObj:=Plywood;
    MoveL Offs(pOrigin,120.40,-66.68,-0.00),v40,z0,tcp\WObj:=Plywood;
    MoveL Offs(pOrigin,120.15,-65.78,-0.00),v40,z0,tcp\WObj:=Plywood;
    MoveL Offs(pOrigin,119.90,-65.78,-0.00),v40,z0,tcp\WObj:=Plywood;
    MoveL Offs(pOrigin,119.75,-66.38,-0.00),v40,z0,tcp\WObj:=Plywood;
    MoveL Offs(pOrigin,120.10,-66.97,-0.00),v40,z0,tcp\WObj:=Plywood;
    MoveL Offs(pOrigin,120.80,-67.43,-0.00),v40,z0,tcp\WObj:=Plywood;
    MoveL Offs(pOrigin,121.25,-67.22,-0.00),v40,z0,tcp\WObj:=Plywood;
    MoveL Offs(pOrigin,121.25,-66.88,-0.00),v40,fine,tcp\WObj:=Plywood;
    MoveL Offs(pOrigin,121.25,-66.88,-6.00),v60,z5,tcp\WObj:=Plywood;
    MoveL Offs(pOrigin,120.25,-65.47,-6.00),vTravel,z5,tcp\WObj:=Plywood;
    MoveL Offs(pOrigin,120.25,-65.47,-0.00),v60,z0,tcp\WObj:=Plywood;
    MoveL Offs(pOrigin,121.60,-65.18,-0.00),v40,z0,tcp\WObj:=Plywood;
    MoveL Offs(pOrigin,120.95,-64.88,-0.00),v40,z0,tcp\WObj:=Plywood;
    MoveL Offs(pOrigin,120.25,-65.47,-0.00),v40,fine,tcp\WObj:=Plywood;
    MoveL Offs(pOrigin,120.25,-65.47,-6.00),v60,z5,tcp\WObj:=Plywood;
    MoveL Offs(pOrigin,116.90,-72.53,-6.00),vTravel,z5,tcp\WObj:=Plywood;
    MoveL Offs(pOrigin,116.90,-72.53,-0.00),v60,z0,tcp\WObj:=Plywood;
    MoveL Offs(pOrigin,116.60,-72.38,-0.00),v40,z0,tcp\WObj:=Plywood;
    MoveL Offs(pOrigin,116.60,-72.82,-0.00),v40,z0,tcp\WObj:=Plywood;
    MoveL Offs(pOrigin,116.90,-72.53,-0.00),v40,z0,tcp\WObj:=Plywood;
    MoveL Offs(pOrigin,116.60,-72.38,-0.00),v40,z0,tcp\WObj:=Plywood;
    MoveL Offs(pOrigin,116.45,-72.68,-0.00),v40,z0,tcp\WObj:=Plywood;
    MoveL Offs(pOrigin,116.90,-72.53,-0.00),v40,z0,tcp\WObj:=Plywood;
    MoveL Offs(pOrigin,116.30,-72.97,-0.00),v40,z0,tcp\WObj:=Plywood;
    MoveL Offs(pOrigin,115.85,-73.28,-0.00),v40,z0,tcp\WObj:=Plywood;
    MoveL Offs(pOrigin,116.30,-73.43,-0.00),v40,z0,tcp\WObj:=Plywood;
    MoveL Offs(pOrigin,116.45,-73.12,-0.00),v40,z0,tcp\WObj:=Plywood;
    MoveL Offs(pOrigin,116.15,-72.97,-0.00),v40,z0,tcp\WObj:=Plywood;
    MoveL Offs(pOrigin,115.85,-73.28,-0.00),v40,z0,tcp\WObj:=Plywood;
    MoveL Offs(pOrigin,116.30,-73.43,-0.00),v40,z0,tcp\WObj:=Plywood;
    MoveL Offs(pOrigin,116.30,-72.97,-0.00),v40,fine,tcp\WObj:=Plywood;
    MoveL Offs(pOrigin,116.30,-72.97,-6.00),v60,z5,tcp\WObj:=Plywood;
    MoveL Offs(pOrigin,117.20,-73.97,-6.00),vTravel,z5,tcp\WObj:=Plywood;
    MoveL Offs(pOrigin,117.20,-73.97,-0.00),v60,z0,tcp\WObj:=Plywood;
    MoveL Offs(pOrigin,116.75,-75.18,-0.00),v40,z0,tcp\WObj:=Plywood;
    MoveL Offs(pOrigin,117.40,-74.47,-0.00),v40,z0,tcp\WObj:=Plywood;
    MoveL Offs(pOrigin,117.20,-73.97,-0.00),v40,z0,tcp\WObj:=Plywood;
    MoveL Offs(pOrigin,117.95,-74.78,-0.00),v40,z0,tcp\WObj:=Plywood;
    MoveL Offs(pOrigin,117.95,-75.22,-0.00),v40,z0,tcp\WObj:=Plywood;
    MoveL Offs(pOrigin,118.25,-74.93,-0.00),v40,z0,tcp\WObj:=Plywood;
    MoveL Offs(pOrigin,117.95,-74.78,-0.00),v40,z0,tcp\WObj:=Plywood;
    MoveL Offs(pOrigin,117.80,-75.07,-0.00),v40,z0,tcp\WObj:=Plywood;
    MoveL Offs(pOrigin,118.25,-74.93,-0.00),v40,z0,tcp\WObj:=Plywood;
    MoveL Offs(pOrigin,117.95,-74.78,-0.00),v40,fine,tcp\WObj:=Plywood;
    MoveL Offs(pOrigin,117.95,-74.78,-6.00),v60,z5,tcp\WObj:=Plywood;
    MoveL Offs(pOrigin,119.00,-75.82,-6.00),vTravel,z5,tcp\WObj:=Plywood;
    MoveL Offs(pOrigin,119.00,-75.82,-0.00),v60,z0,tcp\WObj:=Plywood;
    MoveL Offs(pOrigin,117.65,-77.28,-0.00),v40,z0,tcp\WObj:=Plywood;
    MoveL Offs(pOrigin,118.40,-77.18,-0.00),v40,z0,tcp\WObj:=Plywood;
    MoveL Offs(pOrigin,119.25,-76.43,-0.00),v40,z0,tcp\WObj:=Plywood;
    MoveL Offs(pOrigin,119.40,-75.82,-0.00),v40,z0,tcp\WObj:=Plywood;
    MoveL Offs(pOrigin,119.00,-75.82,-0.00),v40,z0,tcp\WObj:=Plywood;
    MoveL Offs(pOrigin,119.75,-76.72,-0.00),v40,z0,tcp\WObj:=Plywood;
    MoveL Offs(pOrigin,118.65,-77.78,-0.00),v40,z0,tcp\WObj:=Plywood;
    MoveL Offs(pOrigin,118.65,-78.53,-0.00),v40,z0,tcp\WObj:=Plywood;
    MoveL Offs(pOrigin,119.15,-78.93,-0.00),v40,z0,tcp\WObj:=Plywood;
    MoveL Offs(pOrigin,119.00,-78.22,-0.00),v40,z0,tcp\WObj:=Plywood;
    MoveL Offs(pOrigin,119.30,-77.62,-0.00),v40,z0,tcp\WObj:=Plywood;
    MoveL Offs(pOrigin,120.30,-77.47,-0.00),v40,z0,tcp\WObj:=Plywood;
    MoveL Offs(pOrigin,120.50,-77.93,-0.00),v40,z0,tcp\WObj:=Plywood;
    MoveL Offs(pOrigin,120.20,-78.53,-0.00),v40,z0,tcp\WObj:=Plywood;
    MoveL Offs(pOrigin,119.25,-78.97,-0.00),v40,z0,tcp\WObj:=Plywood;
    MoveL Offs(pOrigin,119.75,-79.38,-0.00),v40,z0,tcp\WObj:=Plywood;
    MoveL Offs(pOrigin,121.40,-78.22,-0.00),v40,z0,tcp\WObj:=Plywood;
    MoveL Offs(pOrigin,121.90,-77.47,-0.00),v40,z0,tcp\WObj:=Plywood;
    MoveL Offs(pOrigin,121.75,-76.72,-0.00),v40,z0,tcp\WObj:=Plywood;
    MoveL Offs(pOrigin,121.10,-76.07,-0.00),v40,z0,tcp\WObj:=Plywood;
    MoveL Offs(pOrigin,120.50,-75.97,-0.00),v40,z0,tcp\WObj:=Plywood;
    MoveL Offs(pOrigin,120.25,-76.28,-0.00),v40,z0,tcp\WObj:=Plywood;
    MoveL Offs(pOrigin,120.95,-76.72,-0.00),v40,z0,tcp\WObj:=Plywood;
    MoveL Offs(pOrigin,121.20,-77.32,-0.00),v40,z0,tcp\WObj:=Plywood;
    MoveL Offs(pOrigin,119.75,-76.72,-0.00),v40,fine,tcp\WObj:=Plywood;
    MoveL Offs(pOrigin,119.75,-76.72,-6.00),v60,z5,tcp\WObj:=Plywood;
    MoveL Offs(pOrigin,120.80,-96.53,-6.00),vTravel,z5,tcp\WObj:=Plywood;
    MoveL Offs(pOrigin,120.80,-96.53,-0.00),v60,z0,tcp\WObj:=Plywood;
    MoveL Offs(pOrigin,120.80,-97.12,-0.00),v40,z0,tcp\WObj:=Plywood;
    MoveL Offs(pOrigin,121.25,-96.82,-0.00),v40,z0,tcp\WObj:=Plywood;
  ENDPROC

  PROC DrawPart9()
    MoveL Offs(pOrigin,120.80,-96.53,-0.00),v40,z0,tcp\WObj:=Plywood;
    MoveL Offs(pOrigin,120.65,-96.97,-0.00),v40,z0,tcp\WObj:=Plywood;
    MoveL Offs(pOrigin,120.95,-97.12,-0.00),v40,z0,tcp\WObj:=Plywood;
    MoveL Offs(pOrigin,121.25,-96.68,-0.00),v40,z0,tcp\WObj:=Plywood;
    MoveL Offs(pOrigin,120.80,-96.53,-0.00),v40,fine,tcp\WObj:=Plywood;
    MoveL Offs(pOrigin,120.80,-96.53,-6.00),v60,z5,tcp\WObj:=Plywood;
    MoveL Offs(pOrigin,120.20,-97.57,-6.00),vTravel,z5,tcp\WObj:=Plywood;
    MoveL Offs(pOrigin,120.20,-97.57,-0.00),v60,z0,tcp\WObj:=Plywood;
    MoveL Offs(pOrigin,120.65,-97.28,-0.00),v40,z0,tcp\WObj:=Plywood;
    MoveL Offs(pOrigin,120.20,-97.57,-0.00),v40,z0,tcp\WObj:=Plywood;
    MoveL Offs(pOrigin,120.20,-97.57,-0.00),v40,z0,tcp\WObj:=Plywood;
    MoveL Offs(pOrigin,119.75,-97.88,-0.00),v40,z0,tcp\WObj:=Plywood;
    MoveL Offs(pOrigin,120.05,-98.03,-0.00),v40,z0,tcp\WObj:=Plywood;
    MoveL Offs(pOrigin,120.35,-97.72,-0.00),v40,z0,tcp\WObj:=Plywood;
    MoveL Offs(pOrigin,120.05,-97.57,-0.00),v40,z0,tcp\WObj:=Plywood;
    MoveL Offs(pOrigin,119.75,-97.88,-0.00),v40,z0,tcp\WObj:=Plywood;
    MoveL Offs(pOrigin,120.05,-98.03,-0.00),v40,z0,tcp\WObj:=Plywood;
    MoveL Offs(pOrigin,120.20,-97.57,-0.00),v40,fine,tcp\WObj:=Plywood;
    MoveL Offs(pOrigin,120.20,-97.57,-6.00),v60,z5,tcp\WObj:=Plywood;
    MoveL Offs(pOrigin,121.25,-102.22,-6.00),vTravel,z5,tcp\WObj:=Plywood;
    MoveL Offs(pOrigin,121.25,-102.22,-0.00),v60,z0,tcp\WObj:=Plywood;
    MoveL Offs(pOrigin,120.50,-102.53,-0.00),v40,z0,tcp\WObj:=Plywood;
    MoveL Offs(pOrigin,119.75,-103.43,-0.00),v40,z0,tcp\WObj:=Plywood;
    MoveL Offs(pOrigin,120.05,-104.47,-0.00),v40,z0,tcp\WObj:=Plywood;
    MoveL Offs(pOrigin,120.80,-104.93,-0.00),v40,z0,tcp\WObj:=Plywood;
    MoveL Offs(pOrigin,121.35,-104.47,-0.00),v40,z0,tcp\WObj:=Plywood;
    MoveL Offs(pOrigin,120.40,-104.18,-0.00),v40,z0,tcp\WObj:=Plywood;
    MoveL Offs(pOrigin,120.50,-103.12,-0.00),v40,z0,tcp\WObj:=Plywood;
    MoveL Offs(pOrigin,121.40,-102.88,-0.00),v40,z0,tcp\WObj:=Plywood;
    MoveL Offs(pOrigin,121.85,-103.97,-0.00),v40,z0,tcp\WObj:=Plywood;
    MoveL Offs(pOrigin,122.40,-103.43,-0.00),v40,z0,tcp\WObj:=Plywood;
    MoveL Offs(pOrigin,122.15,-102.82,-0.00),v40,z0,tcp\WObj:=Plywood;
    MoveL Offs(pOrigin,121.25,-102.22,-0.00),v40,fine,tcp\WObj:=Plywood;
    MoveL Offs(pOrigin,121.25,-102.22,-6.00),v60,z5,tcp\WObj:=Plywood;
    MoveL Offs(pOrigin,122.45,-104.03,-6.00),vTravel,z5,tcp\WObj:=Plywood;
    MoveL Offs(pOrigin,122.45,-104.03,-0.00),v60,z0,tcp\WObj:=Plywood;
    MoveL Offs(pOrigin,120.65,-105.82,-0.00),v40,z0,tcp\WObj:=Plywood;
    MoveL Offs(pOrigin,120.55,-106.28,-0.00),v40,z0,tcp\WObj:=Plywood;
    MoveL Offs(pOrigin,120.95,-106.38,-0.00),v40,z0,tcp\WObj:=Plywood;
    MoveL Offs(pOrigin,122.30,-105.22,-0.00),v40,z0,tcp\WObj:=Plywood;
    MoveL Offs(pOrigin,123.05,-104.03,-0.00),v40,z0,tcp\WObj:=Plywood;
    MoveL Offs(pOrigin,122.45,-104.03,-0.00),v40,z0,tcp\WObj:=Plywood;
    MoveL Offs(pOrigin,122.45,-105.22,-0.00),v40,z0,tcp\WObj:=Plywood;
    MoveL Offs(pOrigin,122.00,-105.97,-0.00),v40,z0,tcp\WObj:=Plywood;
    MoveL Offs(pOrigin,122.15,-106.88,-0.00),v40,z0,tcp\WObj:=Plywood;
    MoveL Offs(pOrigin,123.20,-107.62,-0.00),v40,z0,tcp\WObj:=Plywood;
    MoveL Offs(pOrigin,123.95,-107.32,-0.00),v40,z0,tcp\WObj:=Plywood;
    MoveL Offs(pOrigin,124.85,-106.28,-0.00),v40,z0,tcp\WObj:=Plywood;
    MoveL Offs(pOrigin,124.65,-105.38,-0.00),v40,z0,tcp\WObj:=Plywood;
    MoveL Offs(pOrigin,123.80,-104.78,-0.00),v40,z0,tcp\WObj:=Plywood;
    MoveL Offs(pOrigin,122.45,-105.22,-0.00),v40,z0,tcp\WObj:=Plywood;
    MoveL Offs(pOrigin,123.25,-105.53,-0.00),v40,z0,tcp\WObj:=Plywood;
    MoveL Offs(pOrigin,123.65,-105.53,-0.00),v40,z0,tcp\WObj:=Plywood;
    MoveL Offs(pOrigin,124.05,-106.22,-0.00),v40,z0,tcp\WObj:=Plywood;
    MoveL Offs(pOrigin,123.25,-105.53,-0.00),v40,z0,tcp\WObj:=Plywood;
    MoveL Offs(pOrigin,122.80,-106.22,-0.00),v40,z0,tcp\WObj:=Plywood;
    MoveL Offs(pOrigin,123.20,-106.72,-0.00),v40,z0,tcp\WObj:=Plywood;
    MoveL Offs(pOrigin,122.80,-106.68,-0.00),v40,z0,tcp\WObj:=Plywood;
    MoveL Offs(pOrigin,122.80,-106.22,-0.00),v40,fine,tcp\WObj:=Plywood;
    MoveL Offs(pOrigin,122.80,-106.22,-6.00),v60,z5,tcp\WObj:=Plywood;
    MoveL Offs(pOrigin,123.85,-107.78,-6.00),vTravel,z5,tcp\WObj:=Plywood;
    MoveL Offs(pOrigin,123.85,-107.78,-0.00),v60,z0,tcp\WObj:=Plywood;
    MoveL Offs(pOrigin,123.85,-108.68,-0.00),v40,z0,tcp\WObj:=Plywood;
    MoveL Offs(pOrigin,124.55,-109.53,-0.00),v40,z0,tcp\WObj:=Plywood;
    MoveL Offs(pOrigin,125.15,-109.68,-0.00),v40,z0,tcp\WObj:=Plywood;
    MoveL Offs(pOrigin,126.65,-108.38,-0.00),v40,z0,tcp\WObj:=Plywood;
    MoveL Offs(pOrigin,125.35,-110.03,-0.00),v40,z0,tcp\WObj:=Plywood;
    MoveL Offs(pOrigin,126.50,-111.32,-0.00),v40,z0,tcp\WObj:=Plywood;
    MoveL Offs(pOrigin,127.40,-111.32,-0.00),v40,z0,tcp\WObj:=Plywood;
    MoveL Offs(pOrigin,129.20,-109.32,-0.00),v40,z0,tcp\WObj:=Plywood;
    MoveL Offs(pOrigin,128.15,-109.32,-0.00),v40,z0,tcp\WObj:=Plywood;
    MoveL Offs(pOrigin,126.85,-110.43,-0.00),v40,z0,tcp\WObj:=Plywood;
    MoveL Offs(pOrigin,126.70,-109.88,-0.00),v40,z0,tcp\WObj:=Plywood;
    MoveL Offs(pOrigin,127.65,-108.53,-0.00),v40,z0,tcp\WObj:=Plywood;
    MoveL Offs(pOrigin,125.45,-106.32,-0.00),v40,z0,tcp\WObj:=Plywood;
    MoveL Offs(pOrigin,124.85,-106.47,-0.00),v40,z0,tcp\WObj:=Plywood;
    MoveL Offs(pOrigin,123.85,-107.78,-0.00),v40,z0,tcp\WObj:=Plywood;
    MoveL Offs(pOrigin,124.55,-107.78,-0.00),v40,z0,tcp\WObj:=Plywood;
    MoveL Offs(pOrigin,124.85,-108.07,-0.00),v40,z0,tcp\WObj:=Plywood;
    MoveL Offs(pOrigin,124.55,-108.22,-0.00),v40,z0,tcp\WObj:=Plywood;
    MoveL Offs(pOrigin,124.55,-107.78,-0.00),v40,z0,tcp\WObj:=Plywood;
    MoveL Offs(pOrigin,124.85,-108.22,-0.00),v40,z0,tcp\WObj:=Plywood;
    MoveL Offs(pOrigin,124.55,-108.22,-0.00),v40,z0,tcp\WObj:=Plywood;
    MoveL Offs(pOrigin,124.55,-107.78,-0.00),v40,z0,tcp\WObj:=Plywood;
    MoveL Offs(pOrigin,125.30,-107.32,-0.00),v40,z0,tcp\WObj:=Plywood;
    MoveL Offs(pOrigin,125.75,-107.62,-0.00),v40,z0,tcp\WObj:=Plywood;
    MoveL Offs(pOrigin,125.60,-108.07,-0.00),v40,z0,tcp\WObj:=Plywood;
    MoveL Offs(pOrigin,125.30,-107.32,-0.00),v40,z0,tcp\WObj:=Plywood;
    MoveL Offs(pOrigin,125.75,-107.62,-0.00),v40,z0,tcp\WObj:=Plywood;
    MoveL Offs(pOrigin,125.60,-108.07,-0.00),v40,z0,tcp\WObj:=Plywood;
    MoveL Offs(pOrigin,125.30,-107.32,-0.00),v40,fine,tcp\WObj:=Plywood;
    MoveL Offs(pOrigin,125.30,-107.32,-6.00),v60,z5,tcp\WObj:=Plywood;
    MoveL Offs(pOrigin,128.75,-111.47,-6.00),vTravel,z5,tcp\WObj:=Plywood;
    MoveL Offs(pOrigin,128.75,-111.47,-0.00),v60,z0,tcp\WObj:=Plywood;
    MoveL Offs(pOrigin,129.55,-111.53,-0.00),v40,z0,tcp\WObj:=Plywood;
    MoveL Offs(pOrigin,129.35,-112.38,-0.00),v40,z0,tcp\WObj:=Plywood;
    MoveL Offs(pOrigin,128.60,-112.28,-0.00),v40,z0,tcp\WObj:=Plywood;
    MoveL Offs(pOrigin,128.75,-111.47,-0.00),v40,fine,tcp\WObj:=Plywood;
    MoveL Offs(pOrigin,128.75,-111.47,-6.00),v60,z5,tcp\WObj:=Plywood;
    MoveL Offs(pOrigin,131.90,-115.88,-6.00),vTravel,z5,tcp\WObj:=Plywood;
    MoveL Offs(pOrigin,131.90,-115.88,-0.00),v60,z0,tcp\WObj:=Plywood;
    MoveL Offs(pOrigin,132.05,-115.43,-0.00),v40,z0,tcp\WObj:=Plywood;
    MoveL Offs(pOrigin,131.90,-115.88,-0.00),v40,fine,tcp\WObj:=Plywood;
    MoveL Offs(pOrigin,131.90,-115.88,-6.00),v60,z5,tcp\WObj:=Plywood;
    MoveL Offs(pOrigin,137.00,-108.82,-6.00),vTravel,z5,tcp\WObj:=Plywood;
    MoveL Offs(pOrigin,137.00,-108.82,-0.00),v60,z0,tcp\WObj:=Plywood;
    MoveL Offs(pOrigin,137.90,-109.43,-0.00),v40,z0,tcp\WObj:=Plywood;
    MoveL Offs(pOrigin,139.65,-107.93,-0.00),v40,z0,tcp\WObj:=Plywood;
    MoveL Offs(pOrigin,138.20,-106.43,-0.00),v40,z0,tcp\WObj:=Plywood;
    MoveL Offs(pOrigin,137.45,-107.18,-0.00),v40,z0,tcp\WObj:=Plywood;
    MoveL Offs(pOrigin,138.00,-108.53,-0.00),v40,z0,tcp\WObj:=Plywood;
    MoveL Offs(pOrigin,137.50,-108.53,-0.00),v40,z0,tcp\WObj:=Plywood;
    MoveL Offs(pOrigin,137.15,-107.68,-0.00),v40,z0,tcp\WObj:=Plywood;
    MoveL Offs(pOrigin,136.70,-107.93,-0.00),v40,z0,tcp\WObj:=Plywood;
    MoveL Offs(pOrigin,137.00,-108.82,-0.00),v40,fine,tcp\WObj:=Plywood;
    MoveL Offs(pOrigin,137.00,-108.82,-6.00),v60,z5,tcp\WObj:=Plywood;
    MoveL Offs(pOrigin,138.15,-107.78,-6.00),vTravel,z5,tcp\WObj:=Plywood;
    MoveL Offs(pOrigin,138.15,-107.78,-0.00),v60,z0,tcp\WObj:=Plywood;
    MoveL Offs(pOrigin,138.25,-107.22,-0.00),v40,z0,tcp\WObj:=Plywood;
    MoveL Offs(pOrigin,138.70,-107.62,-0.00),v40,z0,tcp\WObj:=Plywood;
  ENDPROC

  PROC DrawPart10()
    MoveL Offs(pOrigin,138.50,-108.07,-0.00),v40,z0,tcp\WObj:=Plywood;
    MoveL Offs(pOrigin,138.15,-107.78,-0.00),v40,fine,tcp\WObj:=Plywood;
    MoveL Offs(pOrigin,138.15,-107.78,-6.00),v60,z5,tcp\WObj:=Plywood;
    MoveL Offs(pOrigin,140.00,-108.47,-6.00),vTravel,z5,tcp\WObj:=Plywood;
    MoveL Offs(pOrigin,140.00,-108.47,-0.00),v60,z0,tcp\WObj:=Plywood;
    MoveL Offs(pOrigin,138.40,-110.03,-0.00),v40,z0,tcp\WObj:=Plywood;
    MoveL Offs(pOrigin,139.55,-111.22,-0.00),v40,z0,tcp\WObj:=Plywood;
    MoveL Offs(pOrigin,140.60,-110.88,-0.00),v40,z0,tcp\WObj:=Plywood;
    MoveL Offs(pOrigin,141.40,-109.88,-0.00),v40,z0,tcp\WObj:=Plywood;
    MoveL Offs(pOrigin,141.20,-109.57,-0.00),v40,z0,tcp\WObj:=Plywood;
    MoveL Offs(pOrigin,140.00,-110.53,-0.00),v40,z0,tcp\WObj:=Plywood;
    MoveL Offs(pOrigin,139.45,-110.47,-0.00),v40,z0,tcp\WObj:=Plywood;
    MoveL Offs(pOrigin,139.45,-109.88,-0.00),v40,z0,tcp\WObj:=Plywood;
    MoveL Offs(pOrigin,140.25,-108.82,-0.00),v40,z0,tcp\WObj:=Plywood;
    MoveL Offs(pOrigin,140.00,-108.47,-0.00),v40,fine,tcp\WObj:=Plywood;
    MoveL Offs(pOrigin,140.00,-108.47,-6.00),v60,z5,tcp\WObj:=Plywood;
    MoveL Offs(pOrigin,142.55,-109.82,-6.00),vTravel,z5,tcp\WObj:=Plywood;
    MoveL Offs(pOrigin,142.55,-109.82,-0.00),v60,z0,tcp\WObj:=Plywood;
    MoveL Offs(pOrigin,140.35,-111.82,-0.00),v40,z0,tcp\WObj:=Plywood;
    MoveL Offs(pOrigin,141.05,-112.88,-0.00),v40,z0,tcp\WObj:=Plywood;
    MoveL Offs(pOrigin,141.65,-113.18,-0.00),v40,z0,tcp\WObj:=Plywood;
    MoveL Offs(pOrigin,142.55,-112.88,-0.00),v40,z0,tcp\WObj:=Plywood;
    MoveL Offs(pOrigin,143.30,-111.68,-0.00),v40,z0,tcp\WObj:=Plywood;
    MoveL Offs(pOrigin,142.85,-111.18,-0.00),v40,z0,tcp\WObj:=Plywood;
    MoveL Offs(pOrigin,142.55,-112.38,-0.00),v40,z0,tcp\WObj:=Plywood;
    MoveL Offs(pOrigin,141.80,-112.72,-0.00),v40,z0,tcp\WObj:=Plywood;
    MoveL Offs(pOrigin,141.25,-112.28,-0.00),v40,z0,tcp\WObj:=Plywood;
    MoveL Offs(pOrigin,141.80,-111.22,-0.00),v40,z0,tcp\WObj:=Plywood;
    MoveL Offs(pOrigin,142.55,-111.03,-0.00),v40,z0,tcp\WObj:=Plywood;
    MoveL Offs(pOrigin,142.55,-109.82,-0.00),v40,fine,tcp\WObj:=Plywood;
    MoveL Offs(pOrigin,142.55,-109.82,-6.00),v60,z5,tcp\WObj:=Plywood;
    MoveL Offs(pOrigin,143.60,-112.62,-6.00),vTravel,z5,tcp\WObj:=Plywood;
    MoveL Offs(pOrigin,143.60,-112.62,-0.00),v60,z0,tcp\WObj:=Plywood;
    MoveL Offs(pOrigin,142.40,-113.88,-0.00),v40,z0,tcp\WObj:=Plywood;
    MoveL Offs(pOrigin,142.85,-113.93,-0.00),v40,z0,tcp\WObj:=Plywood;
    MoveL Offs(pOrigin,143.60,-112.62,-0.00),v40,fine,tcp\WObj:=Plywood;
    MoveL Offs(pOrigin,143.60,-112.62,-6.00),v60,z5,tcp\WObj:=Plywood;
    MoveL Offs(pOrigin,143.15,-114.38,-6.00),vTravel,z5,tcp\WObj:=Plywood;
    MoveL Offs(pOrigin,143.15,-114.38,-0.00),v60,z0,tcp\WObj:=Plywood;
    MoveL Offs(pOrigin,143.15,-114.82,-0.00),v40,z0,tcp\WObj:=Plywood;
    MoveL Offs(pOrigin,143.60,-114.68,-0.00),v40,z0,tcp\WObj:=Plywood;
    MoveL Offs(pOrigin,143.00,-114.53,-0.00),v40,z0,tcp\WObj:=Plywood;
    MoveL Offs(pOrigin,143.15,-114.82,-0.00),v40,z0,tcp\WObj:=Plywood;
    MoveL Offs(pOrigin,143.60,-114.68,-0.00),v40,z0,tcp\WObj:=Plywood;
    MoveL Offs(pOrigin,143.15,-114.38,-0.00),v40,fine,tcp\WObj:=Plywood;
    MoveL Offs(pOrigin,143.15,-114.38,-6.00),v60,z5,tcp\WObj:=Plywood;
    MoveL Offs(pOrigin,136.10,-106.78,-6.00),vTravel,z5,tcp\WObj:=Plywood;
    MoveL Offs(pOrigin,136.10,-106.78,-0.00),v60,z0,tcp\WObj:=Plywood;
    MoveL Offs(pOrigin,135.55,-106.57,-0.00),v40,z0,tcp\WObj:=Plywood;
    MoveL Offs(pOrigin,135.65,-106.18,-0.00),v40,z0,tcp\WObj:=Plywood;
    MoveL Offs(pOrigin,136.10,-106.43,-0.00),v40,z0,tcp\WObj:=Plywood;
    MoveL Offs(pOrigin,136.10,-106.78,-0.00),v40,fine,tcp\WObj:=Plywood;
    MoveL Offs(pOrigin,136.10,-106.78,-6.00),v60,z5,tcp\WObj:=Plywood;
    MoveL Offs(pOrigin,121.80,-114.22,-6.00),vTravel,z5,tcp\WObj:=Plywood;
    MoveL Offs(pOrigin,121.80,-114.22,-0.00),v60,z0,tcp\WObj:=Plywood;
    MoveL Offs(pOrigin,121.10,-113.57,-0.00),v40,z0,tcp\WObj:=Plywood;
    MoveL Offs(pOrigin,120.50,-113.47,-0.00),v40,z0,tcp\WObj:=Plywood;
    MoveL Offs(pOrigin,120.20,-113.78,-0.00),v40,z0,tcp\WObj:=Plywood;
    MoveL Offs(pOrigin,121.10,-114.38,-0.00),v40,z0,tcp\WObj:=Plywood;
    MoveL Offs(pOrigin,121.20,-114.82,-0.00),v40,z0,tcp\WObj:=Plywood;
    MoveL Offs(pOrigin,119.75,-114.22,-0.00),v40,z0,tcp\WObj:=Plywood;
    MoveL Offs(pOrigin,118.65,-115.28,-0.00),v40,z0,tcp\WObj:=Plywood;
    MoveL Offs(pOrigin,118.55,-115.72,-0.00),v40,z0,tcp\WObj:=Plywood;
    MoveL Offs(pOrigin,119.00,-116.38,-0.00),v40,z0,tcp\WObj:=Plywood;
    MoveL Offs(pOrigin,119.30,-115.12,-0.00),v40,z0,tcp\WObj:=Plywood;
    MoveL Offs(pOrigin,119.90,-114.82,-0.00),v40,z0,tcp\WObj:=Plywood;
    MoveL Offs(pOrigin,120.35,-114.97,-0.00),v40,z0,tcp\WObj:=Plywood;
    MoveL Offs(pOrigin,120.50,-115.43,-0.00),v40,z0,tcp\WObj:=Plywood;
    MoveL Offs(pOrigin,120.20,-116.03,-0.00),v40,z0,tcp\WObj:=Plywood;
    MoveL Offs(pOrigin,119.25,-116.47,-0.00),v40,z0,tcp\WObj:=Plywood;
    MoveL Offs(pOrigin,119.75,-116.88,-0.00),v40,z0,tcp\WObj:=Plywood;
    MoveL Offs(pOrigin,121.75,-115.28,-0.00),v40,z0,tcp\WObj:=Plywood;
    MoveL Offs(pOrigin,121.80,-114.22,-0.00),v40,fine,tcp\WObj:=Plywood;
    MoveL Offs(pOrigin,121.80,-114.22,-6.00),v60,z5,tcp\WObj:=Plywood;
    MoveL Offs(pOrigin,119.30,-113.93,-6.00),vTravel,z5,tcp\WObj:=Plywood;
    MoveL Offs(pOrigin,119.30,-113.93,-0.00),v60,z0,tcp\WObj:=Plywood;
    MoveL Offs(pOrigin,119.40,-113.32,-0.00),v40,z0,tcp\WObj:=Plywood;
    MoveL Offs(pOrigin,119.00,-113.32,-0.00),v40,z0,tcp\WObj:=Plywood;
    MoveL Offs(pOrigin,117.65,-114.78,-0.00),v40,z0,tcp\WObj:=Plywood;
    MoveL Offs(pOrigin,118.25,-114.72,-0.00),v40,z0,tcp\WObj:=Plywood;
    MoveL Offs(pOrigin,119.30,-113.93,-0.00),v40,fine,tcp\WObj:=Plywood;
    MoveL Offs(pOrigin,119.30,-113.93,-6.00),v60,z5,tcp\WObj:=Plywood;
    MoveL Offs(pOrigin,117.30,-112.12,-6.00),vTravel,z5,tcp\WObj:=Plywood;
    MoveL Offs(pOrigin,117.30,-112.12,-0.00),v60,z0,tcp\WObj:=Plywood;
    MoveL Offs(pOrigin,117.20,-111.62,-0.00),v40,z0,tcp\WObj:=Plywood;
    MoveL Offs(pOrigin,116.90,-112.53,-0.00),v40,z0,tcp\WObj:=Plywood;
    MoveL Offs(pOrigin,117.30,-112.12,-0.00),v40,fine,tcp\WObj:=Plywood;
    MoveL Offs(pOrigin,117.30,-112.12,-6.00),v60,z5,tcp\WObj:=Plywood;
    MoveL Offs(pOrigin,116.30,-110.93,-6.00),vTravel,z5,tcp\WObj:=Plywood;
    MoveL Offs(pOrigin,116.30,-110.93,-0.00),v60,z0,tcp\WObj:=Plywood;
    MoveL Offs(pOrigin,116.45,-110.62,-0.00),v40,z0,tcp\WObj:=Plywood;
    MoveL Offs(pOrigin,116.00,-110.78,-0.00),v40,z0,tcp\WObj:=Plywood;
    MoveL Offs(pOrigin,116.30,-110.93,-0.00),v40,z0,tcp\WObj:=Plywood;
    MoveL Offs(pOrigin,116.30,-110.47,-0.00),v40,z0,tcp\WObj:=Plywood;
    MoveL Offs(pOrigin,116.00,-110.78,-0.00),v40,z0,tcp\WObj:=Plywood;
    MoveL Offs(pOrigin,116.30,-110.93,-0.00),v40,fine,tcp\WObj:=Plywood;
    MoveL Offs(pOrigin,116.30,-110.93,-6.00),v60,z5,tcp\WObj:=Plywood;
    MoveL Offs(pOrigin,174.55,-92.97,-6.00),vTravel,z5,tcp\WObj:=Plywood;
    MoveL Offs(pOrigin,174.55,-92.97,-0.00),v60,z0,tcp\WObj:=Plywood;
    MoveL Offs(pOrigin,199.20,-93.12,-0.00),v40,z0,tcp\WObj:=Plywood;
    MoveL Offs(pOrigin,199.25,-102.53,-0.00),v40,z0,tcp\WObj:=Plywood;
    MoveL Offs(pOrigin,198.20,-102.28,-0.00),v40,z0,tcp\WObj:=Plywood;
    MoveL Offs(pOrigin,197.15,-103.12,-0.00),v40,z0,tcp\WObj:=Plywood;
    MoveL Offs(pOrigin,197.00,-103.88,-0.00),v40,z0,tcp\WObj:=Plywood;
    MoveL Offs(pOrigin,197.75,-104.78,-0.00),v40,z0,tcp\WObj:=Plywood;
    MoveL Offs(pOrigin,198.35,-104.93,-0.00),v40,z0,tcp\WObj:=Plywood;
    MoveL Offs(pOrigin,198.70,-104.62,-0.00),v40,z0,tcp\WObj:=Plywood;
    MoveL Offs(pOrigin,197.80,-104.12,-0.00),v40,z0,tcp\WObj:=Plywood;
    MoveL Offs(pOrigin,197.80,-103.28,-0.00),v40,z0,tcp\WObj:=Plywood;
    MoveL Offs(pOrigin,198.35,-102.82,-0.00),v40,z0,tcp\WObj:=Plywood;
    MoveL Offs(pOrigin,199.25,-103.28,-0.00),v40,z0,tcp\WObj:=Plywood;
    MoveL Offs(pOrigin,199.20,-104.78,-0.00),v40,z0,tcp\WObj:=Plywood;
    MoveL Offs(pOrigin,197.90,-106.12,-0.00),v40,z0,tcp\WObj:=Plywood;
    MoveL Offs(pOrigin,198.35,-106.43,-0.00),v40,z0,tcp\WObj:=Plywood;
    MoveL Offs(pOrigin,199.25,-105.53,-0.00),v40,z0,tcp\WObj:=Plywood;
    MoveL Offs(pOrigin,199.35,-133.07,-0.00),v40,z0,tcp\WObj:=Plywood;
    MoveL Offs(pOrigin,174.50,-133.07,-0.00),v40,z0,tcp\WObj:=Plywood;
    MoveL Offs(pOrigin,174.55,-92.97,-0.00),v40,fine,tcp\WObj:=Plywood;
    MoveL Offs(pOrigin,174.55,-92.97,-6.00),v60,z5,tcp\WObj:=Plywood;
    MoveL Offs(pOrigin,174.55,-90.32,-6.00),vTravel,z5,tcp\WObj:=Plywood;
  ENDPROC

  PROC DrawPart11()
    MoveL Offs(pOrigin,174.55,-90.32,-0.00),v60,z0,tcp\WObj:=Plywood;
    MoveL Offs(pOrigin,174.40,-50.92,-0.00),v40,z0,tcp\WObj:=Plywood;
    MoveL Offs(pOrigin,199.35,-50.83,-0.00),v40,z0,tcp\WObj:=Plywood;
    MoveL Offs(pOrigin,199.25,-67.12,-0.00),v40,z0,tcp\WObj:=Plywood;
    MoveL Offs(pOrigin,197.90,-68.62,-0.00),v40,z0,tcp\WObj:=Plywood;
    MoveL Offs(pOrigin,198.35,-68.88,-0.00),v40,z0,tcp\WObj:=Plywood;
    MoveL Offs(pOrigin,199.25,-68.03,-0.00),v40,z0,tcp\WObj:=Plywood;
    MoveL Offs(pOrigin,199.20,-90.32,-0.00),v40,z0,tcp\WObj:=Plywood;
    MoveL Offs(pOrigin,191.75,-90.38,-0.00),v40,z0,tcp\WObj:=Plywood;
    MoveL Offs(pOrigin,191.15,-90.12,-0.00),v40,z0,tcp\WObj:=Plywood;
    MoveL Offs(pOrigin,190.40,-90.38,-0.00),v40,z0,tcp\WObj:=Plywood;
    MoveL Offs(pOrigin,189.95,-89.62,-0.00),v40,z0,tcp\WObj:=Plywood;
    MoveL Offs(pOrigin,188.75,-90.38,-0.00),v40,z0,tcp\WObj:=Plywood;
    MoveL Offs(pOrigin,174.55,-90.32,-0.00),v40,fine,tcp\WObj:=Plywood;
    MoveL Offs(pOrigin,174.55,-90.32,-6.00),v60,z5,tcp\WObj:=Plywood;
    MoveL Offs(pOrigin,186.95,-86.93,-6.00),vTravel,z5,tcp\WObj:=Plywood;
    MoveL Offs(pOrigin,186.95,-86.93,-0.00),v60,z0,tcp\WObj:=Plywood;
    MoveL Offs(pOrigin,187.25,-87.07,-0.00),v40,z0,tcp\WObj:=Plywood;
    MoveL Offs(pOrigin,187.40,-86.78,-0.00),v40,z0,tcp\WObj:=Plywood;
    MoveL Offs(pOrigin,186.95,-86.93,-0.00),v40,z0,tcp\WObj:=Plywood;
    MoveL Offs(pOrigin,187.25,-87.07,-0.00),v40,z0,tcp\WObj:=Plywood;
    MoveL Offs(pOrigin,187.25,-86.62,-0.00),v40,z0,tcp\WObj:=Plywood;
    MoveL Offs(pOrigin,186.95,-86.93,-0.00),v40,fine,tcp\WObj:=Plywood;
    MoveL Offs(pOrigin,186.95,-86.93,-6.00),v60,z5,tcp\WObj:=Plywood;
    MoveL Offs(pOrigin,188.15,-87.68,-6.00),vTravel,z5,tcp\WObj:=Plywood;
    MoveL Offs(pOrigin,188.15,-87.68,-0.00),v60,z0,tcp\WObj:=Plywood;
    MoveL Offs(pOrigin,188.00,-88.28,-0.00),v40,z0,tcp\WObj:=Plywood;
    MoveL Offs(pOrigin,188.45,-88.12,-0.00),v40,z0,tcp\WObj:=Plywood;
    MoveL Offs(pOrigin,188.15,-87.68,-0.00),v40,z0,tcp\WObj:=Plywood;
    MoveL Offs(pOrigin,188.15,-88.43,-0.00),v40,z0,tcp\WObj:=Plywood;
    MoveL Offs(pOrigin,188.45,-88.12,-0.00),v40,z0,tcp\WObj:=Plywood;
    MoveL Offs(pOrigin,188.15,-87.68,-0.00),v40,fine,tcp\WObj:=Plywood;
    MoveL Offs(pOrigin,188.15,-87.68,-6.00),v60,z5,tcp\WObj:=Plywood;
    MoveL Offs(pOrigin,189.35,-88.12,-6.00),vTravel,z5,tcp\WObj:=Plywood;
    MoveL Offs(pOrigin,189.35,-88.12,-0.00),v60,z0,tcp\WObj:=Plywood;
    MoveL Offs(pOrigin,189.25,-88.72,-0.00),v40,z0,tcp\WObj:=Plywood;
    MoveL Offs(pOrigin,189.90,-87.97,-0.00),v40,z0,tcp\WObj:=Plywood;
    MoveL Offs(pOrigin,189.35,-88.12,-0.00),v40,fine,tcp\WObj:=Plywood;
    MoveL Offs(pOrigin,189.35,-88.12,-6.00),v60,z5,tcp\WObj:=Plywood;
    MoveL Offs(pOrigin,190.40,-89.18,-6.00),vTravel,z5,tcp\WObj:=Plywood;
    MoveL Offs(pOrigin,190.40,-89.18,-0.00),v60,z0,tcp\WObj:=Plywood;
    MoveL Offs(pOrigin,190.85,-89.47,-0.00),v40,z0,tcp\WObj:=Plywood;
    MoveL Offs(pOrigin,190.85,-89.03,-0.00),v40,z0,tcp\WObj:=Plywood;
    MoveL Offs(pOrigin,190.40,-89.32,-0.00),v40,z0,tcp\WObj:=Plywood;
    MoveL Offs(pOrigin,190.85,-89.47,-0.00),v40,z0,tcp\WObj:=Plywood;
    MoveL Offs(pOrigin,191.00,-89.18,-0.00),v40,z0,tcp\WObj:=Plywood;
    MoveL Offs(pOrigin,190.40,-89.18,-0.00),v40,fine,tcp\WObj:=Plywood;
    MoveL Offs(pOrigin,190.40,-89.18,-6.00),v60,z5,tcp\WObj:=Plywood;
    MoveL Offs(pOrigin,193.05,-94.12,-6.00),vTravel,z5,tcp\WObj:=Plywood;
    MoveL Offs(pOrigin,193.05,-94.12,-0.00),v60,z0,tcp\WObj:=Plywood;
    MoveL Offs(pOrigin,193.85,-94.28,-0.00),v40,z0,tcp\WObj:=Plywood;
    MoveL Offs(pOrigin,194.20,-93.97,-0.00),v40,z0,tcp\WObj:=Plywood;
    MoveL Offs(pOrigin,193.05,-94.12,-0.00),v40,fine,tcp\WObj:=Plywood;
    MoveL Offs(pOrigin,193.05,-94.12,-6.00),v60,z5,tcp\WObj:=Plywood;
    MoveL Offs(pOrigin,194.15,-94.88,-6.00),vTravel,z5,tcp\WObj:=Plywood;
    MoveL Offs(pOrigin,194.15,-94.88,-0.00),v60,z0,tcp\WObj:=Plywood;
    MoveL Offs(pOrigin,194.60,-94.57,-0.00),v40,z0,tcp\WObj:=Plywood;
    MoveL Offs(pOrigin,194.15,-94.88,-0.00),v40,z0,tcp\WObj:=Plywood;
    MoveL Offs(pOrigin,194.90,-93.97,-0.00),v40,z0,tcp\WObj:=Plywood;
    MoveL Offs(pOrigin,195.20,-94.12,-0.00),v40,z0,tcp\WObj:=Plywood;
    MoveL Offs(pOrigin,195.35,-93.82,-0.00),v40,z0,tcp\WObj:=Plywood;
    MoveL Offs(pOrigin,194.90,-93.97,-0.00),v40,z0,tcp\WObj:=Plywood;
    MoveL Offs(pOrigin,195.20,-94.12,-0.00),v40,z0,tcp\WObj:=Plywood;
    MoveL Offs(pOrigin,195.20,-93.68,-0.00),v40,z0,tcp\WObj:=Plywood;
    MoveL Offs(pOrigin,194.90,-93.97,-0.00),v40,z0,tcp\WObj:=Plywood;
    MoveL Offs(pOrigin,194.45,-93.68,-0.00),v40,z0,tcp\WObj:=Plywood;
    MoveL Offs(pOrigin,194.45,-93.22,-0.00),v40,z0,tcp\WObj:=Plywood;
    MoveL Offs(pOrigin,194.45,-93.68,-0.00),v40,fine,tcp\WObj:=Plywood;
    MoveL Offs(pOrigin,194.45,-93.68,-6.00),v60,z5,tcp\WObj:=Plywood;
    MoveL Offs(pOrigin,196.55,-94.78,-6.00),vTravel,z5,tcp\WObj:=Plywood;
    MoveL Offs(pOrigin,196.55,-94.78,-0.00),v60,z0,tcp\WObj:=Plywood;
    MoveL Offs(pOrigin,194.75,-96.07,-0.00),v40,z0,tcp\WObj:=Plywood;
    MoveL Offs(pOrigin,195.65,-95.93,-0.00),v40,z0,tcp\WObj:=Plywood;
    MoveL Offs(pOrigin,196.55,-94.78,-0.00),v40,z0,tcp\WObj:=Plywood;
    MoveL Offs(pOrigin,197.00,-95.62,-0.00),v40,z0,tcp\WObj:=Plywood;
    MoveL Offs(pOrigin,196.65,-95.93,-0.00),v40,z0,tcp\WObj:=Plywood;
    MoveL Offs(pOrigin,197.35,-95.78,-0.00),v40,z0,tcp\WObj:=Plywood;
    MoveL Offs(pOrigin,197.00,-95.62,-0.00),v40,z0,tcp\WObj:=Plywood;
    MoveL Offs(pOrigin,196.55,-95.93,-0.00),v40,z0,tcp\WObj:=Plywood;
    MoveL Offs(pOrigin,196.25,-96.22,-0.00),v40,z0,tcp\WObj:=Plywood;
    MoveL Offs(pOrigin,196.40,-96.53,-0.00),v40,z0,tcp\WObj:=Plywood;
    MoveL Offs(pOrigin,196.70,-96.07,-0.00),v40,z0,tcp\WObj:=Plywood;
    MoveL Offs(pOrigin,196.25,-96.22,-0.00),v40,z0,tcp\WObj:=Plywood;
    MoveL Offs(pOrigin,196.40,-96.53,-0.00),v40,z0,tcp\WObj:=Plywood;
    MoveL Offs(pOrigin,196.70,-96.22,-0.00),v40,z0,tcp\WObj:=Plywood;
    MoveL Offs(pOrigin,196.55,-95.93,-0.00),v40,z0,tcp\WObj:=Plywood;
    MoveL Offs(pOrigin,196.25,-96.47,-0.00),v40,z0,tcp\WObj:=Plywood;
    MoveL Offs(pOrigin,196.00,-96.82,-0.00),v40,z0,tcp\WObj:=Plywood;
    MoveL Offs(pOrigin,196.25,-97.32,-0.00),v40,z0,tcp\WObj:=Plywood;
    MoveL Offs(pOrigin,196.25,-96.47,-0.00),v40,fine,tcp\WObj:=Plywood;
    MoveL Offs(pOrigin,196.25,-96.47,-6.00),v60,z5,tcp\WObj:=Plywood;
    MoveL Offs(pOrigin,196.90,-98.03,-6.00),vTravel,z5,tcp\WObj:=Plywood;
    MoveL Offs(pOrigin,196.90,-98.03,-0.00),v60,z0,tcp\WObj:=Plywood;
    MoveL Offs(pOrigin,197.45,-98.03,-0.00),v40,z0,tcp\WObj:=Plywood;
    MoveL Offs(pOrigin,198.60,-96.68,-0.00),v40,z0,tcp\WObj:=Plywood;
    MoveL Offs(pOrigin,198.20,-96.68,-0.00),v40,z0,tcp\WObj:=Plywood;
    MoveL Offs(pOrigin,196.90,-98.03,-0.00),v40,fine,tcp\WObj:=Plywood;
    MoveL Offs(pOrigin,196.90,-98.03,-6.00),v60,z5,tcp\WObj:=Plywood;
    MoveL Offs(pOrigin,202.25,-93.12,-6.00),vTravel,z5,tcp\WObj:=Plywood;
    MoveL Offs(pOrigin,202.25,-93.12,-0.00),v60,z0,tcp\WObj:=Plywood;
    MoveL Offs(pOrigin,227.25,-92.97,-0.00),v40,z0,tcp\WObj:=Plywood;
    MoveL Offs(pOrigin,223.55,-96.97,-0.00),v40,z0,tcp\WObj:=Plywood;
    MoveL Offs(pOrigin,217.50,-101.18,-0.00),v40,z0,tcp\WObj:=Plywood;
    MoveL Offs(pOrigin,221.75,-105.38,-0.00),v40,z0,tcp\WObj:=Plywood;
    MoveL Offs(pOrigin,223.50,-108.22,-0.00),v40,z0,tcp\WObj:=Plywood;
    MoveL Offs(pOrigin,224.75,-111.97,-0.00),v40,z0,tcp\WObj:=Plywood;
    MoveL Offs(pOrigin,225.05,-114.22,-0.00),v40,z0,tcp\WObj:=Plywood;
    MoveL Offs(pOrigin,224.75,-119.32,-0.00),v40,z0,tcp\WObj:=Plywood;
    MoveL Offs(pOrigin,223.90,-122.03,-0.00),v40,z0,tcp\WObj:=Plywood;
    MoveL Offs(pOrigin,222.25,-125.18,-0.00),v40,z0,tcp\WObj:=Plywood;
    MoveL Offs(pOrigin,219.20,-128.77,-0.00),v40,z0,tcp\WObj:=Plywood;
    MoveL Offs(pOrigin,216.65,-130.62,-0.00),v40,z0,tcp\WObj:=Plywood;
    MoveL Offs(pOrigin,213.65,-132.12,-0.00),v40,z0,tcp\WObj:=Plywood;
    MoveL Offs(pOrigin,209.30,-133.12,-0.00),v40,z0,tcp\WObj:=Plywood;
    MoveL Offs(pOrigin,202.10,-133.07,-0.00),v40,z0,tcp\WObj:=Plywood;
    MoveL Offs(pOrigin,202.25,-109.57,-0.00),v40,z0,tcp\WObj:=Plywood;
    MoveL Offs(pOrigin,204.05,-107.93,-0.00),v40,z0,tcp\WObj:=Plywood;
    MoveL Offs(pOrigin,203.45,-107.03,-0.00),v40,z0,tcp\WObj:=Plywood;
    MoveL Offs(pOrigin,202.25,-106.43,-0.00),v40,z0,tcp\WObj:=Plywood;
    MoveL Offs(pOrigin,202.25,-93.12,-0.00),v40,fine,tcp\WObj:=Plywood;
  ENDPROC

